  MoveL 1327 to (239.11, 156.17, 31.63) mm, rotated rx -180 ry 0 rz 180 deg; joints [-146.664, -89.82, -20.414, 62.265, 38.38, -56.149]
  MoveL 1328 to (239.11, 156.17, 31.63) mm, rotated rx -180 ry 0 rz 180 deg; joints [-146.664, -89.82, -20.414, 62.265, 38.38, -56.149]
  Call Extruder(256.49281)
  MoveL 1329 to (239, 156.42, 31.63) mm, rotated rx -180 ry 0 rz -180 deg; joints [-146.64, -89.832, -20.39, 62.3, 38.394, -56.183]
  MoveL 1330 to (239, 156.42, 31.63) mm, rotated rx -180 ry 0 rz -180 deg; joints [-146.64, -89.832, -20.39, 62.3, 38.394, -56.183]
  Call Extruder(256.65113)
  MoveL 1331 to (238.89, 156.66, 31.63) mm, rotated rx -180 ry 0 rz 180 deg; joints [-146.617, -89.843, -20.367, 62.335, 38.409, -56.217]
  MoveL 1332 to (238.89, 156.66, 31.63) mm, rotated rx -180 ry 0 rz 180 deg; joints [-146.617, -89.843, -20.367, 62.335, 38.409, -56.217]
  Call Extruder(256.83316)
  MoveL 1333 to (238.75, 156.94, 31.63) mm, rotated rx 180 ry 0 rz 180 deg; joints [-146.589, -89.851, -20.35, 62.369, 38.428, -56.249]
  MoveL 1334 to (238.75, 156.94, 31.63) mm, rotated rx 180 ry 0 rz 180 deg; joints [-146.589, -89.851, -20.35, 62.369, 38.428, -56.249]
  Call Extruder(257.03972)
  MoveL 1335 to (238.57, 157.25, 31.63) mm, rotated rx 180 ry 0 rz 180 deg; joints [-146.557, -89.857, -20.339, 62.403, 38.451, -56.278]
  MoveL 1336 to (238.57, 157.25, 31.63) mm, rotated rx 180 ry 0 rz 180 deg; joints [-146.557, -89.857, -20.339, 62.403, 38.451, -56.278]
  Call Extruder(257.24706)
  MoveL 1337 to (238.4, 157.55, 31.63) mm, rotated rx -180 ry 0 rz 180 deg; joints [-146.526, -89.862, -20.328, 62.437, 38.475, -56.308]
  MoveL 1338 to (238.4, 157.55, 31.63) mm, rotated rx -180 ry 0 rz 180 deg; joints [-146.526, -89.862, -20.328, 62.437, 38.475, -56.308]
  Call Extruder(257.45518)
  MoveL 1339 to (238.22, 157.85, 31.63) mm, rotated rx -180 ry 0 rz 180 deg; joints [-146.495, -89.867, -20.318, 62.471, 38.499, -56.338]
  MoveL 1340 to (238.22, 157.85, 31.63) mm, rotated rx -180 ry 0 rz 180 deg; joints [-146.495, -89.867, -20.318, 62.471, 38.499, -56.338]
  Call Extruder(257.57289)
  MoveL 1341 to (238.12, 158.03, 31.63) mm, rotated rx 180 ry 0 rz 180 deg; joints [-146.477, -89.87, -20.312, 62.49, 38.512, -56.354]
  MoveL 1342 to (238.12, 158.03, 31.63) mm, rotated rx 180 ry 0 rz 180 deg; joints [-146.477, -89.87, -20.312, 62.49, 38.512, -56.354]
  Call Extruder(257.90571)
  MoveL 1343 to (237.79, 158.48, 31.63) mm, rotated rx 180 ry 0 rz 180 deg; joints [-146.427, -89.864, -20.324, 62.528, 38.557, -56.38]
  MoveL 1344 to (237.79, 158.48, 31.63) mm, rotated rx 180 ry 0 rz 180 deg; joints [-146.427, -89.864, -20.324, 62.528, 38.557, -56.38]
  Call Extruder(258.23971)
  MoveL 1345 to (237.47, 158.93, 31.63) mm, rotated rx -180 ry 0 rz 180 deg; joints [-146.377, -89.858, -20.336, 62.566, 38.601, -56.406]
  MoveL 1346 to (237.47, 158.93, 31.63) mm, rotated rx -180 ry 0 rz 180 deg; joints [-146.377, -89.858, -20.336, 62.566, 38.601, -56.406]
  Call Extruder(258.40729)
  MoveL 1347 to (237.3, 159.15, 31.63) mm, rotated rx 180 ry 0 rz -180 deg; joints [-146.352, -89.855, -20.341, 62.585, 38.623, -56.419]
  Call Extruder(259.23663)
  MoveL 1348 to (236.39, 160.19, 31.63) mm, rotated rx 180 ry 0 rz 180 deg; joints [-146.229, -89.811, -20.432, 62.642, 38.747, -56.438]
  Call Extruder(259.86767)
  MoveL 1349 to (235.61, 160.89, 31.63) mm, rotated rx 180 ry 0 rz -180 deg; joints [-146.138, -89.747, -20.564, 62.648, 38.854, -56.406]
  MoveL 1350 to (235.61, 160.89, 31.63) mm, rotated rx 180 ry 0 rz -180 deg; joints [-146.138, -89.747, -20.564, 62.648, 38.854, -56.406]
  Call Extruder(260.06527)
  MoveL 1351 to (235.35, 161.1, 31.63) mm, rotated rx 180 ry 0 rz 180 deg; joints [-146.109, -89.725, -20.608, 62.648, 38.888, -56.394]
  Call Extruder(260.39930)
  MoveL 1352 to (234.9, 161.43, 31.63) mm, rotated rx 180 ry 0 rz -180 deg; joints [-146.062, -89.679, -20.702, 62.637, 38.949, -56.357]
  MoveL 1353 to (234.9, 161.43, 31.63) mm, rotated rx 180 ry 0 rz -180 deg; joints [-146.062, -89.679, -20.702, 62.637, 38.949, -56.357]
  Call Extruder(260.73214)
  MoveL 1354 to (234.45, 161.76, 31.63) mm, rotated rx 180 ry 0 rz 180 deg; joints [-146.015, -89.633, -20.796, 62.625, 39.01, -56.322]
  MoveL 1355 to (234.45, 161.76, 31.63) mm, rotated rx 180 ry 0 rz 180 deg; joints [-146.015, -89.633, -20.796, 62.625, 39.01, -56.322]
  Call Extruder(260.91134)
  MoveL 1356 to (234.21, 161.93, 31.63) mm, rotated rx -180 ry 0 rz 180 deg; joints [-145.99, -89.608, -20.848, 62.619, 39.044, -56.302]
  MoveL 1357 to (234.21, 161.93, 31.63) mm, rotated rx -180 ry 0 rz 180 deg; joints [-145.99, -89.608, -20.848, 62.619, 39.044, -56.302]
  Call Extruder(261.11946)
  MoveL 1358 to (233.9, 162.11, 31.63) mm, rotated rx 180 ry 0 rz 180 deg; joints [-145.961, -89.572, -20.923, 62.602, 39.085, -56.267]
  MoveL 1359 to (233.9, 162.11, 31.63) mm, rotated rx 180 ry 0 rz 180 deg; joints [-145.961, -89.572, -20.923, 62.602, 39.085, -56.267]
  Call Extruder(261.32679)
  MoveL 1360 to (233.6, 162.29, 31.63) mm, rotated rx 180 ry 0 rz 180 deg; joints [-145.933, -89.535, -20.998, 62.585, 39.126, -56.232]
  MoveL 1361 to (233.6, 162.29, 31.63) mm, rotated rx 180 ry 0 rz 180 deg; joints [-145.933, -89.535, -20.998, 62.585, 39.126, -56.232]
  Call Extruder(261.53335)
  MoveL 1362 to (233.29, 162.46, 31.63) mm, rotated rx -180 ry 0 rz -180 deg; joints [-145.905, -89.498, -21.073, 62.568, 39.167, -56.198]
  MoveL 1363 to (233.29, 162.46, 31.63) mm, rotated rx -180 ry 0 rz -180 deg; joints [-145.905, -89.498, -21.073, 62.568, 39.167, -56.198]
  Call Extruder(261.73913)
  MoveL 1364 to (232.99, 162.64, 31.63) mm, rotated rx 180 ry 0 rz -180 deg; joints [-145.876, -89.462, -21.147, 62.551, 39.209, -56.164]
  MoveL 1365 to (232.99, 162.64, 31.63) mm, rotated rx 180 ry 0 rz -180 deg; joints [-145.876, -89.462, -21.147, 62.551, 39.209, -56.164]
  Call Extruder(261.89741)
  MoveL 1366 to (232.74, 162.74, 31.63) mm, rotated rx -180 ry 0 rz 180 deg; joints [-145.856, -89.427, -21.218, 62.53, 39.242, -56.127]
  MoveL 1367 to (232.74, 162.74, 31.63) mm, rotated rx -180 ry 0 rz 180 deg; joints [-145.856, -89.427, -21.218, 62.53, 39.242, -56.127]
  Call Extruder(262.05508)
  MoveL 1368 to (232.49, 162.85, 31.63) mm, rotated rx 180 ry 0 rz -180 deg; joints [-145.835, -89.393, -21.289, 62.508, 39.276, -56.09]
  MoveL 1369 to (232.49, 162.85, 31.63) mm, rotated rx 180 ry 0 rz -180 deg; joints [-145.835, -89.393, -21.289, 62.508, 39.276, -56.09]
  Call Extruder(262.22517)
  MoveL 1370 to (232.22, 162.97, 31.63) mm, rotated rx 180 ry 0 rz 180 deg; joints [-145.813, -89.355, -21.366, 62.485, 39.313, -56.049]
  MoveL 1371 to (232.22, 162.97, 31.63) mm, rotated rx 180 ry 0 rz 180 deg; joints [-145.813, -89.355, -21.366, 62.485, 39.313, -56.049]
  Call Extruder(262.40753)
  MoveL 1372 to (231.93, 163.09, 31.63) mm, rotated rx -180 ry 0 rz 180 deg; joints [-145.789, -89.314, -21.45, 62.46, 39.352, -56.005]
  MoveL 1373 to (231.93, 163.09, 31.63) mm, rotated rx -180 ry 0 rz 180 deg; joints [-145.789, -89.314, -21.45, 62.46, 39.352, -56.005]
  Call Extruder(262.58914)
  MoveL 1374 to (231.64, 163.21, 31.63) mm, rotated rx -180 ry 0 rz 180 deg; joints [-145.766, -89.274, -21.534, 62.434, 39.392, -55.962]
  MoveL 1375 to (231.64, 163.21, 31.63) mm, rotated rx -180 ry 0 rz 180 deg; joints [-145.766, -89.274, -21.534, 62.434, 39.392, -55.962]
  Call Extruder(262.70258)
  MoveL 1376 to (231.45, 163.27, 31.63) mm, rotated rx 180 ry 0 rz -180 deg; joints [-145.751, -89.245, -21.592, 62.415, 39.417, -55.93]
  MoveL 1377 to (231.45, 163.27, 31.63) mm, rotated rx 180 ry 0 rz -180 deg; joints [-145.751, -89.245, -21.592, 62.415, 39.417, -55.93]
  Call Extruder(262.81558)
  MoveL 1378 to (231.26, 163.33, 31.63) mm, rotated rx 180 ry 0 rz 180 deg; joints [-145.737, -89.217, -21.65, 62.395, 39.443, -55.898]
  MoveL 1379 to (231.26, 163.33, 31.63) mm, rotated rx 180 ry 0 rz 180 deg; joints [-145.737, -89.217, -21.65, 62.395, 39.443, -55.898]
  Call Extruder(262.92814)
  MoveL 1380 to (231.07, 163.39, 31.63) mm, rotated rx -180 ry 0 rz -180 deg; joints [-145.723, -89.189, -21.708, 62.375, 39.468, -55.866]
  MoveL 1381 to (231.07, 163.39, 31.63) mm, rotated rx -180 ry 0 rz -180 deg; joints [-145.723, -89.189, -21.708, 62.375, 39.468, -55.866]
  Call Extruder(263.04025)
  MoveL 1382 to (230.88, 163.45, 31.63) mm, rotated rx 180 ry 0 rz 180 deg; joints [-145.709, -89.16, -21.766, 62.356, 39.494, -55.834]
  MoveL 1383 to (230.88, 163.45, 31.63) mm, rotated rx 180 ry 0 rz 180 deg; joints [-145.709, -89.16, -21.766, 62.356, 39.494, -55.834]
  Call Extruder(263.15191)
  MoveL 1384 to (230.7, 163.51, 31.63) mm, rotated rx 180 ry 0 rz -180 deg; joints [-145.695, -89.132, -21.824, 62.336, 39.519, -55.802]
  MoveL 1385 to (230.7, 163.51, 31.63) mm, rotated rx 180 ry 0 rz -180 deg; joints [-145.695, -89.132, -21.824, 62.336, 39.519, -55.802]
  Call Extruder(263.28301)
  MoveL 1386 to (230.47, 163.58, 31.63) mm, rotated rx 180 ry 0 rz 180 deg; joints [-145.679, -89.098, -21.894, 62.312, 39.55, -55.764]
  MoveL 1387 to (230.47, 163.58, 31.63) mm, rotated rx 180 ry 0 rz 180 deg; joints [-145.679, -89.098, -21.894, 62.312, 39.55, -55.764]
  Call Extruder(263.41354)
  MoveL 1388 to (230.25, 163.65, 31.63) mm, rotated rx -180 ry 0 rz 180 deg; joints [-145.662, -89.064, -21.964, 62.288, 39.58, -55.725]
  MoveL 1389 to (230.25, 163.65, 31.63) mm, rotated rx -180 ry 0 rz 180 deg; joints [-145.662, -89.064, -21.964, 62.288, 39.58, -55.725]
  Call Extruder(263.54350)
  MoveL 1390 to (230.02, 163.72, 31.63) mm, rotated rx 180 ry 0 rz 180 deg; joints [-145.646, -89.031, -22.033, 62.265, 39.61, -55.687]
  MoveL 1391 to (230.02, 163.72, 31.63) mm, rotated rx 180 ry 0 rz 180 deg; joints [-145.646, -89.031, -22.033, 62.265, 39.61, -55.687]
  Call Extruder(263.67290)
  MoveL 1392 to (229.8, 163.78, 31.63) mm, rotated rx -180 ry 0 rz 180 deg; joints [-145.629, -88.997, -22.102, 62.241, 39.64, -55.648]
  MoveL 1393 to (229.8, 163.78, 31.63) mm, rotated rx -180 ry 0 rz 180 deg; joints [-145.629, -88.997, -22.102, 62.241, 39.64, -55.648]
  Call Extruder(263.79488)
  MoveL 1394 to (229.59, 163.84, 31.63) mm, rotated rx 180 ry 0 rz -180 deg; joints [-145.614, -88.964, -22.171, 62.217, 39.669, -55.61]
  MoveL 1395 to (229.59, 163.84, 31.63) mm, rotated rx 180 ry 0 rz -180 deg; joints [-145.614, -88.964, -22.171, 62.217, 39.669, -55.61]
  Call Extruder(263.90973)
  MoveL 1396 to (229.38, 163.88, 31.63) mm, rotated rx 180 ry 0 rz -180 deg; joints [-145.601, -88.931, -22.238, 62.192, 39.696, -55.571]
  MoveL 1397 to (229.38, 163.88, 31.63) mm, rotated rx 180 ry 0 rz -180 deg; joints [-145.601, -88.931, -22.238, 62.192, 39.696, -55.571]
  Call Extruder(264.02412)
  MoveL 1398 to (229.18, 163.93, 31.63) mm, rotated rx 180 ry 0 rz -180 deg; joints [-145.587, -88.898, -22.306, 62.167, 39.724, -55.533]
  MoveL 1399 to (229.18, 163.93, 31.63) mm, rotated rx 180 ry 0 rz -180 deg; joints [-145.587, -88.898, -22.306, 62.167, 39.724, -55.533]
  Call Extruder(264.13806)
  MoveL 1400 to (228.97, 163.97, 31.63) mm, rotated rx 180 ry 0 rz 180 deg; joints [-145.573, -88.865, -22.373, 62.143, 39.751, -55.494]
  MoveL 1401 to (228.97, 163.97, 31.63) mm, rotated rx 180 ry 0 rz 180 deg; joints [-145.573, -88.865, -22.373, 62.143, 39.751, -55.494]
  Call Extruder(264.25155)
  MoveL 1402 to (228.77, 164.02, 31.63) mm, rotated rx -180 ry 0 rz 180 deg; joints [-145.559, -88.833, -22.44, 62.118, 39.779, -55.456]
  MoveL 1403 to (228.77, 164.02, 31.63) mm, rotated rx -180 ry 0 rz 180 deg; joints [-145.559, -88.833, -22.44, 62.118, 39.779, -55.456]
  Call Extruder(264.38884)
  MoveL 1404 to (228.52, 164.07, 31.63) mm, rotated rx -180 ry 0 rz -180 deg; joints [-145.543, -88.792, -22.523, 62.088, 39.812, -55.408]
  MoveL 1405 to (228.52, 164.07, 31.63) mm, rotated rx -180 ry 0 rz -180 deg; joints [-145.543, -88.792, -22.523, 62.088, 39.812, -55.408]
  Call Extruder(264.52551)
  MoveL 1406 to (228.27, 164.12, 31.63) mm, rotated rx -180 ry 0 rz 180 deg; joints [-145.527, -88.752, -22.606, 62.057, 39.846, -55.36]
  MoveL 1407 to (228.27, 164.12, 31.63) mm, rotated rx -180 ry 0 rz 180 deg; joints [-145.527, -88.752, -22.606, 62.057, 39.846, -55.36]
  Call Extruder(264.66157)
  MoveL 1408 to (228.02, 164.17, 31.63) mm, rotated rx -180 ry 0 rz -180 deg; joints [-145.51, -88.712, -22.689, 62.027, 39.879, -55.313]
  MoveL 1409 to (228.02, 164.17, 31.63) mm, rotated rx -180 ry 0 rz -180 deg; joints [-145.51, -88.712, -22.689, 62.027, 39.879, -55.313]
  Call Extruder(264.79703)
  MoveL 1410 to (227.77, 164.22, 31.63) mm, rotated rx 180 ry 0 rz -180 deg; joints [-145.494, -88.672, -22.771, 61.996, 39.913, -55.266]
  MoveL 1411 to (227.77, 164.22, 31.63) mm, rotated rx 180 ry 0 rz -180 deg; joints [-145.494, -88.672, -22.771, 61.996, 39.913, -55.266]
  Call Extruder(264.93187)
  MoveL 1412 to (227.52, 164.27, 31.63) mm, rotated rx 180 ry 0 rz -180 deg; joints [-145.477, -88.632, -22.853, 61.966, 39.946, -55.219]
  MoveL 1413 to (227.52, 164.27, 31.63) mm, rotated rx 180 ry 0 rz -180 deg; joints [-145.477, -88.632, -22.853, 61.966, 39.946, -55.219]
  Call Extruder(265.06610)
  MoveL 1414 to (227.27, 164.32, 31.63) mm, rotated rx -180 ry 0 rz 180 deg; joints [-145.461, -88.593, -22.935, 61.937, 39.979, -55.172]
  MoveL 1415 to (227.27, 164.32, 31.63) mm, rotated rx -180 ry 0 rz 180 deg; joints [-145.461, -88.593, -22.935, 61.937, 39.979, -55.172]
  Call Extruder(265.19972)
  MoveL 1416 to (227.02, 164.37, 31.63) mm, rotated rx 180 ry 0 rz -180 deg; joints [-145.444, -88.553, -23.017, 61.907, 40.013, -55.125]
  MoveL 1417 to (227.02, 164.37, 31.63) mm, rotated rx 180 ry 0 rz -180 deg; joints [-145.444, -88.553, -23.017, 61.907, 40.013, -55.125]
  Call Extruder(265.36183)
  MoveL 1418 to (226.72, 164.41, 31.63) mm, rotated rx -180 ry 0 rz 180 deg; joints [-145.425, -88.503, -23.12, 61.868, 40.054, -55.066]
  MoveL 1419 to (226.72, 164.41, 31.63) mm, rotated rx -180 ry 0 rz 180 deg; joints [-145.425, -88.503, -23.12, 61.868, 40.054, -55.066]
  Call Extruder(265.52320)
  MoveL 1420 to (226.41, 164.46, 31.63) mm, rotated rx 180 ry 0 rz 180 deg; joints [-145.406, -88.453, -23.223, 61.83, 40.094, -55.006]
  MoveL 1421 to (226.41, 164.46, 31.63) mm, rotated rx 180 ry 0 rz 180 deg; joints [-145.406, -88.453, -23.223, 61.83, 40.094, -55.006]
  Call Extruder(265.68385)
  MoveL 1422 to (226.11, 164.51, 31.63) mm, rotated rx 180 ry 0 rz 180 deg; joints [-145.386, -88.403, -23.326, 61.792, 40.135, -54.947]
  MoveL 1423 to (226.11, 164.51, 31.63) mm, rotated rx 180 ry 0 rz 180 deg; joints [-145.386, -88.403, -23.326, 61.792, 40.135, -54.947]
  Call Extruder(265.84377)
  MoveL 1424 to (225.8, 164.56, 31.63) mm, rotated rx -180 ry 0 rz 180 deg; joints [-145.367, -88.354, -23.428, 61.754, 40.176, -54.888]
  MoveL 1425 to (225.8, 164.56, 31.63) mm, rotated rx -180 ry 0 rz 180 deg; joints [-145.367, -88.354, -23.428, 61.754, 40.176, -54.888]
  Call Extruder(266.00296)
  MoveL 1426 to (225.5, 164.61, 31.63) mm, rotated rx 180 ry 0 rz 180 deg; joints [-145.348, -88.304, -23.53, 61.717, 40.217, -54.83]
  MoveL 1427 to (225.5, 164.61, 31.63) mm, rotated rx 180 ry 0 rz 180 deg; joints [-145.348, -88.304, -23.53, 61.717, 40.217, -54.83]
  Call Extruder(266.16143)
  MoveL 1428 to (225.19, 164.66, 31.63) mm, rotated rx -180 ry 0 rz -180 deg; joints [-145.328, -88.255, -23.632, 61.679, 40.258, -54.771]
  MoveL 1429 to (225.19, 164.66, 31.63) mm, rotated rx -180 ry 0 rz -180 deg; joints [-145.328, -88.255, -23.632, 61.679, 40.258, -54.771]
  Call Extruder(266.36030)
  MoveL 1430 to (224.8, 164.7, 31.63) mm, rotated rx -180 ry 0 rz 180 deg; joints [-145.305, -88.191, -23.764, 61.629, 40.309, -54.694]
  MoveL 1431 to (224.8, 164.7, 31.63) mm, rotated rx -180 ry 0 rz 180 deg; joints [-145.305, -88.191, -23.764, 61.629, 40.309, -54.694]
  Call Extruder(266.55831)
  MoveL 1432 to (224.42, 164.75, 31.63) mm, rotated rx -180 ry 0 rz 180 deg; joints [-145.281, -88.127, -23.896, 61.58, 40.361, -54.618]
  MoveL 1433 to (224.42, 164.75, 31.63) mm, rotated rx -180 ry 0 rz 180 deg; joints [-145.281, -88.127, -23.896, 61.58, 40.361, -54.618]
  Call Extruder(266.75545)
  MoveL 1434 to (224.03, 164.79, 31.63) mm, rotated rx 180 ry 0 rz 180 deg; joints [-145.258, -88.064, -24.027, 61.53, 40.412, -54.542]
  MoveL 1435 to (224.03, 164.79, 31.63) mm, rotated rx 180 ry 0 rz 180 deg; joints [-145.258, -88.064, -24.027, 61.53, 40.412, -54.542]
  Call Extruder(266.95173)
  MoveL 1436 to (223.64, 164.84, 31.63) mm, rotated rx -180 ry 0 rz 180 deg; joints [-145.234, -88, -24.158, 61.482, 40.463, -54.466]
  MoveL 1437 to (223.64, 164.84, 31.63) mm, rotated rx -180 ry 0 rz 180 deg; joints [-145.234, -88, -24.158, 61.482, 40.463, -54.466]
  Call Extruder(267.19740)
  MoveL 1438 to (223.15, 164.89, 31.63) mm, rotated rx 180 ry 0 rz 180 deg; joints [-145.206, -87.92, -24.325, 61.419, 40.528, -54.369]
  MoveL 1439 to (223.15, 164.89, 31.63) mm, rotated rx 180 ry 0 rz 180 deg; joints [-145.206, -87.92, -24.325, 61.419, 40.528, -54.369]
  Call Extruder(267.49209)
  MoveL 1440 to (222.56, 164.93, 31.63) mm, rotated rx -180 ry 0 rz 180 deg; joints [-145.172, -87.821, -24.528, 61.341, 40.606, -54.25]
  MoveL 1441 to (222.56, 164.93, 31.63) mm, rotated rx -180 ry 0 rz 180 deg; joints [-145.172, -87.821, -24.528, 61.341, 40.606, -54.25]
  Call Extruder(267.78545)
  MoveL 1442 to (221.97, 164.98, 31.63) mm, rotated rx 180 ry 0 rz -180 deg; joints [-145.138, -87.724, -24.73, 61.265, 40.684, -54.133]
  MoveL 1443 to (221.97, 164.98, 31.63) mm, rotated rx 180 ry 0 rz -180 deg; joints [-145.138, -87.724, -24.73, 61.265, 40.684, -54.133]
  Call Extruder(268.21876)
  MoveL 1444 to (221.1, 165.02, 31.63) mm, rotated rx -180 ry 0 rz 180 deg; joints [-145.088, -87.578, -25.034, 61.15, 40.799, -53.955]
  MoveL 1445 to (221.1, 165.02, 31.63) mm, rotated rx -180 ry 0 rz 180 deg; joints [-145.088, -87.578, -25.034, 61.15, 40.799, -53.955]
  Call Extruder(268.79092)
  MoveL 1446 to (219.94, 165.07, 31.63) mm, rotated rx 180 ry 0 rz -180 deg; joints [-145.024, -87.384, -25.436, 60.996, 40.952, -53.72]
  MoveL 1447 to (219.94, 165.07, 31.63) mm, rotated rx 180 ry 0 rz -180 deg; joints [-145.024, -87.384, -25.436, 60.996, 40.952, -53.72]
  Call Extruder(269.21879)
  MoveL 1448 to (219.06, 165.09, 31.63) mm, rotated rx -180 ry 0 rz -180 deg; joints [-144.977, -87.238, -25.74, 60.88, 41.066, -53.542]
  Call Extruder(385.86744)
  MoveL 1449 to (-19.06, 165.09, 31.63) mm, rotated rx -180 ry 0 rz -180 deg; joints [-127.435, -66.78, -72.976, 59.702, 66.877, -33.904]
  MoveL 1450 to (-19.06, 165.09, 31.63) mm, rotated rx -180 ry 0 rz -180 deg; joints [-127.435, -66.78, -72.976, 59.702, 66.877, -33.904]
  Call Extruder(386.58306)
  MoveL 1451 to (-20.52, 165.05, 31.63) mm, rotated rx -180 ry 0 rz 180 deg; joints [-127.291, -66.713, -73.159, 59.788, 67.016, -33.846]
  MoveL 1452 to (-20.52, 165.05, 31.63) mm, rotated rx -180 ry 0 rz 180 deg; joints [-127.291, -66.713, -73.159, 59.788, 67.016, -33.846]
  Call Extruder(387.15780)
  MoveL 1453 to (-21.68, 165, 31.63) mm, rotated rx -180 ry 0 rz 180 deg; joints [-127.178, -66.659, -73.307, 59.856, 67.126, -33.797]
  MoveL 1454 to (-21.68, 165, 31.63) mm, rotated rx -180 ry 0 rz 180 deg; joints [-127.178, -66.659, -73.307, 59.856, 67.126, -33.797]
  Call Extruder(387.45117)
  MoveL 1455 to (-22.27, 164.95, 31.63) mm, rotated rx -180 ry 0 rz -180 deg; joints [-127.122, -66.63, -73.386, 59.889, 67.182, -33.77]
  MoveL 1456 to (-22.27, 164.95, 31.63) mm, rotated rx -180 ry 0 rz -180 deg; joints [-127.122, -66.63, -73.386, 59.889, 67.182, -33.77]
  Call Extruder(387.74586)
  MoveL 1457 to (-22.86, 164.91, 31.63) mm, rotated rx 180 ry 0 rz -180 deg; joints [-127.065, -66.602, -73.464, 59.921, 67.239, -33.743]
  MoveL 1458 to (-22.86, 164.91, 31.63) mm, rotated rx 180 ry 0 rz -180 deg; joints [-127.065, -66.602, -73.464, 59.921, 67.239, -33.743]
  Call Extruder(388.04189)
  MoveL 1459 to (-23.45, 164.86, 31.63) mm, rotated rx 180 ry 0 rz 180 deg; joints [-127.009, -66.573, -73.542, 59.954, 67.295, -33.716]
  MoveL 1460 to (-23.45, 164.86, 31.63) mm, rotated rx 180 ry 0 rz 180 deg; joints [-127.009, -66.573, -73.542, 59.954, 67.295, -33.716]
  Call Extruder(388.23816)
  MoveL 1461 to (-23.84, 164.82, 31.63) mm, rotated rx 180 ry 0 rz 180 deg; joints [-126.973, -66.554, -73.596, 59.974, 67.332, -33.696]
  MoveL 1462 to (-23.84, 164.82, 31.63) mm, rotated rx 180 ry 0 rz 180 deg; joints [-126.973, -66.554, -73.596, 59.974, 67.332, -33.696]
  Call Extruder(388.43530)
  MoveL 1463 to (-24.22, 164.77, 31.63) mm, rotated rx 180 ry 0 rz 180 deg; joints [-126.937, -66.535, -73.649, 59.994, 67.369, -33.676]
  MoveL 1464 to (-24.22, 164.77, 31.63) mm, rotated rx 180 ry 0 rz 180 deg; joints [-126.937, -66.535, -73.649, 59.994, 67.369, -33.676]
  Call Extruder(388.63331)
  MoveL 1465 to (-24.61, 164.72, 31.63) mm, rotated rx -180 ry 0 rz 180 deg; joints [-126.901, -66.515, -73.703, 60.014, 67.406, -33.657]
  MoveL 1466 to (-24.61, 164.72, 31.63) mm, rotated rx -180 ry 0 rz 180 deg; joints [-126.901, -66.515, -73.703, 60.014, 67.406, -33.657]
  Call Extruder(388.83219)
  MoveL 1467 to (-25, 164.68, 31.63) mm, rotated rx 180 ry 0 rz 180 deg; joints [-126.865, -66.496, -73.757, 60.034, 67.443, -33.637]
  MoveL 1468 to (-25, 164.68, 31.63) mm, rotated rx 180 ry 0 rz 180 deg; joints [-126.865, -66.496, -73.757, 60.034, 67.443, -33.637]
  Call Extruder(389.01127)
  MoveL 1469 to (-25.34, 164.63, 31.63) mm, rotated rx -180 ry 0 rz -180 deg; joints [-126.834, -66.478, -73.805, 60.051, 67.476, -33.619]
  MoveL 1470 to (-25.34, 164.63, 31.63) mm, rotated rx -180 ry 0 rz -180 deg; joints [-126.834, -66.478, -73.805, 60.051, 67.476, -33.619]
  Call Extruder(389.17046)
  MoveL 1471 to (-25.65, 164.58, 31.63) mm, rotated rx -180 ry 0 rz -180 deg; joints [-126.806, -66.462, -73.85, 60.066, 67.505, -33.602]
  MoveL 1472 to (-25.65, 164.58, 31.63) mm, rotated rx -180 ry 0 rz -180 deg; joints [-126.806, -66.462, -73.85, 60.066, 67.505, -33.602]
  Call Extruder(389.33039)
  MoveL 1473 to (-25.96, 164.53, 31.63) mm, rotated rx 180 ry 0 rz 180 deg; joints [-126.779, -66.446, -73.894, 60.081, 67.535, -33.585]
  MoveL 1474 to (-25.96, 164.53, 31.63) mm, rotated rx 180 ry 0 rz 180 deg; joints [-126.779, -66.446, -73.894, 60.081, 67.535, -33.585]
  Call Extruder(389.49104)
  MoveL 1475 to (-26.26, 164.49, 31.63) mm, rotated rx -180 ry 0 rz 180 deg; joints [-126.751, -66.43, -73.938, 60.096, 67.564, -33.568]
  MoveL 1476 to (-26.26, 164.49, 31.63) mm, rotated rx -180 ry 0 rz 180 deg; joints [-126.751, -66.43, -73.938, 60.096, 67.564, -33.568]
  Call Extruder(389.65242)
  MoveL 1477 to (-26.57, 164.44, 31.63) mm, rotated rx 180 ry 0 rz 180 deg; joints [-126.723, -66.414, -73.982, 60.111, 67.593, -33.551]
  MoveL 1478 to (-26.57, 164.44, 31.63) mm, rotated rx 180 ry 0 rz 180 deg; joints [-126.723, -66.414, -73.982, 60.111, 67.593, -33.551]
  Call Extruder(389.81452)
  MoveL 1479 to (-26.87, 164.39, 31.63) mm, rotated rx -180 ry 0 rz 180 deg; joints [-126.696, -66.399, -74.026, 60.125, 67.622, -33.534]
  MoveL 1480 to (-26.87, 164.39, 31.63) mm, rotated rx -180 ry 0 rz 180 deg; joints [-126.696, -66.399, -74.026, 60.125, 67.622, -33.534]
  Call Extruder(389.96273)
  MoveL 1481 to (-27.15, 164.34, 31.63) mm, rotated rx 180 ry 0 rz 180 deg; joints [-126.671, -66.384, -74.066, 60.138, 67.649, -33.519]
  MoveL 1482 to (-27.15, 164.34, 31.63) mm, rotated rx 180 ry 0 rz 180 deg; joints [-126.671, -66.384, -74.066, 60.138, 67.649, -33.519]
  Call Extruder(390.09696)
  MoveL 1483 to (-27.4, 164.29, 31.63) mm, rotated rx 180 ry 0 rz 180 deg; joints [-126.649, -66.37, -74.104, 60.149, 67.673, -33.504]
  MoveL 1484 to (-27.4, 164.29, 31.63) mm, rotated rx 180 ry 0 rz 180 deg; joints [-126.649, -66.37, -74.104, 60.149, 67.673, -33.504]
  Call Extruder(390.23180)
  MoveL 1485 to (-27.65, 164.24, 31.63) mm, rotated rx -180 ry 0 rz -180 deg; joints [-126.628, -66.357, -74.141, 60.161, 67.697, -33.489]
  MoveL 1486 to (-27.65, 164.24, 31.63) mm, rotated rx -180 ry 0 rz -180 deg; joints [-126.628, -66.357, -74.141, 60.161, 67.697, -33.489]
  Call Extruder(390.36725)
  MoveL 1487 to (-27.9, 164.19, 31.63) mm, rotated rx 180 ry 0 rz 180 deg; joints [-126.606, -66.344, -74.178, 60.172, 67.721, -33.474]
  MoveL 1488 to (-27.9, 164.19, 31.63) mm, rotated rx 180 ry 0 rz 180 deg; joints [-126.606, -66.344, -74.178, 60.172, 67.721, -33.474]
  Call Extruder(390.50331)
  MoveL 1489 to (-28.15, 164.14, 31.63) mm, rotated rx 180 ry 0 rz -180 deg; joints [-126.584, -66.33, -74.216, 60.183, 67.745, -33.459]
  MoveL 1490 to (-28.15, 164.14, 31.63) mm, rotated rx 180 ry 0 rz -180 deg; joints [-126.584, -66.33, -74.216, 60.183, 67.745, -33.459]
  Call Extruder(390.63999)
  MoveL 1491 to (-28.4, 164.09, 31.63) mm, rotated rx 180 ry 0 rz 180 deg; joints [-126.562, -66.317, -74.253, 60.194, 67.769, -33.444]
  MoveL 1492 to (-28.4, 164.09, 31.63) mm, rotated rx 180 ry 0 rz 180 deg; joints [-126.562, -66.317, -74.253, 60.194, 67.769, -33.444]
  Call Extruder(390.77727)
  MoveL 1493 to (-28.64, 164.04, 31.63) mm, rotated rx 180 ry 0 rz 180 deg; joints [-126.54, -66.303, -74.29, 60.206, 67.792, -33.429]
  MoveL 1494 to (-28.64, 164.04, 31.63) mm, rotated rx 180 ry 0 rz 180 deg; joints [-126.54, -66.303, -74.29, 60.206, 67.792, -33.429]
  Call Extruder(390.90294)
  MoveL 1495 to (-28.87, 164, 31.63) mm, rotated rx 180 ry 0 rz 180 deg; joints [-126.52, -66.291, -74.324, 60.216, 67.814, -33.415]
  MoveL 1496 to (-28.87, 164, 31.63) mm, rotated rx 180 ry 0 rz 180 deg; joints [-126.52, -66.291, -74.324, 60.216, 67.814, -33.415]
  Call Extruder(391.01688)
  MoveL 1497 to (-29.08, 163.95, 31.63) mm, rotated rx 180 ry 0 rz 180 deg; joints [-126.503, -66.28, -74.355, 60.224, 67.834, -33.403]
  MoveL 1498 to (-29.08, 163.95, 31.63) mm, rotated rx 180 ry 0 rz 180 deg; joints [-126.503, -66.28, -74.355, 60.224, 67.834, -33.403]
  Call Extruder(391.13127)
  MoveL 1499 to (-29.28, 163.91, 31.63) mm, rotated rx 180 ry 0 rz 180 deg; joints [-126.485, -66.269, -74.386, 60.233, 67.853, -33.39]
  MoveL 1500 to (-29.28, 163.91, 31.63) mm, rotated rx 180 ry 0 rz 180 deg; joints [-126.485, -66.269, -74.386, 60.233, 67.853, -33.39]
  Call Extruder(391.24612)
  MoveL 1501 to (-29.48, 163.86, 31.63) mm, rotated rx 180 ry 0 rz 180 deg; joints [-126.467, -66.258, -74.417, 60.242, 67.873, -33.377]
  MoveL 1502 to (-29.48, 163.86, 31.63) mm, rotated rx 180 ry 0 rz 180 deg; joints [-126.467, -66.258, -74.417, 60.242, 67.873, -33.377]
  Call Extruder(391.36141)
  MoveL 1503 to (-29.69, 163.82, 31.63) mm, rotated rx 180 ry 0 rz 180 deg; joints [-126.45, -66.246, -74.449, 60.251, 67.893, -33.365]
  MoveL 1504 to (-29.69, 163.82, 31.63) mm, rotated rx 180 ry 0 rz 180 deg; joints [-126.45, -66.246, -74.449, 60.251, 67.893, -33.365]
  Call Extruder(391.49081)
  MoveL 1505 to (-29.91, 163.75, 31.63) mm, rotated rx -180 ry 0 rz 180 deg; joints [-126.432, -66.233, -74.485, 60.259, 67.914, -33.349]
  MoveL 1506 to (-29.91, 163.75, 31.63) mm, rotated rx -180 ry 0 rz 180 deg; joints [-126.432, -66.233, -74.485, 60.259, 67.914, -33.349]
  Call Extruder(391.62077)
  MoveL 1507 to (-30.14, 163.68, 31.63) mm, rotated rx 180 ry 0 rz 180 deg; joints [-126.414, -66.22, -74.522, 60.267, 67.936, -33.332]
  MoveL 1508 to (-30.14, 163.68, 31.63) mm, rotated rx 180 ry 0 rz 180 deg; joints [-126.414, -66.22, -74.522, 60.267, 67.936, -33.332]
  Call Extruder(391.75130)
  MoveL 1509 to (-30.36, 163.61, 31.63) mm, rotated rx 180 ry 0 rz 180 deg; joints [-126.396, -66.207, -74.559, 60.275, 67.958, -33.316]
  MoveL 1510 to (-30.36, 163.61, 31.63) mm, rotated rx 180 ry 0 rz 180 deg; joints [-126.396, -66.207, -74.559, 60.275, 67.958, -33.316]
  Call Extruder(391.88239)
  MoveL 1511 to (-30.58, 163.55, 31.63) mm, rotated rx 180 ry 0 rz 180 deg; joints [-126.378, -66.194, -74.596, 60.283, 67.979, -33.3]
  MoveL 1512 to (-30.58, 163.55, 31.63) mm, rotated rx 180 ry 0 rz 180 deg; joints [-126.378, -66.194, -74.596, 60.283, 67.979, -33.3]
  Call Extruder(392.00403)
  MoveL 1513 to (-30.79, 163.48, 31.63) mm, rotated rx 180 ry 0 rz 180 deg; joints [-126.361, -66.181, -74.631, 60.29, 67.999, -33.285]
  MoveL 1514 to (-30.79, 163.48, 31.63) mm, rotated rx 180 ry 0 rz 180 deg; joints [-126.361, -66.181, -74.631, 60.29, 67.999, -33.285]
  Call Extruder(392.11615)
  MoveL 1515 to (-30.98, 163.42, 31.63) mm, rotated rx 180 ry 0 rz -180 deg; joints [-126.347, -66.17, -74.662, 60.296, 68.017, -33.271]
  MoveL 1516 to (-30.98, 163.42, 31.63) mm, rotated rx 180 ry 0 rz -180 deg; joints [-126.347, -66.17, -74.662, 60.296, 68.017, -33.271]
  Call Extruder(392.22871)
  MoveL 1517 to (-31.17, 163.36, 31.63) mm, rotated rx 180 ry 0 rz -180 deg; joints [-126.332, -66.159, -74.694, 60.302, 68.036, -33.257]
  MoveL 1518 to (-31.17, 163.36, 31.63) mm, rotated rx 180 ry 0 rz -180 deg; joints [-126.332, -66.159, -74.694, 60.302, 68.036, -33.257]
  Call Extruder(392.34171)
  MoveL 1519 to (-31.35, 163.3, 31.63) mm, rotated rx 180 ry 0 rz 180 deg; joints [-126.317, -66.147, -74.726, 60.309, 68.054, -33.243]
  MoveL 1520 to (-31.35, 163.3, 31.63) mm, rotated rx 180 ry 0 rz 180 deg; joints [-126.317, -66.147, -74.726, 60.309, 68.054, -33.243]
  Call Extruder(392.45516)
  MoveL 1521 to (-31.54, 163.24, 31.63) mm, rotated rx 180 ry 0 rz 180 deg; joints [-126.302, -66.136, -74.757, 60.315, 68.072, -33.229]
  MoveL 1522 to (-31.54, 163.24, 31.63) mm, rotated rx 180 ry 0 rz 180 deg; joints [-126.302, -66.136, -74.757, 60.315, 68.072, -33.229]
  Call Extruder(392.60280)
  MoveL 1523 to (-31.78, 163.15, 31.63) mm, rotated rx 180 ry 0 rz 180 deg; joints [-126.284, -66.121, -74.8, 60.322, 68.095, -33.209]
  MoveL 1524 to (-31.78, 163.15, 31.63) mm, rotated rx 180 ry 0 rz 180 deg; joints [-126.284, -66.121, -74.8, 60.322, 68.095, -33.209]
  Call Extruder(392.78516)
  MoveL 1525 to (-32.07, 163.03, 31.63) mm, rotated rx 180 ry 0 rz 180 deg; joints [-126.263, -66.102, -74.853, 60.329, 68.124, -33.185]
  MoveL 1526 to (-32.07, 163.03, 31.63) mm, rotated rx 180 ry 0 rz 180 deg; joints [-126.263, -66.102, -74.853, 60.329, 68.124, -33.185]
  Call Extruder(392.96827)
  MoveL 1527 to (-32.37, 162.91, 31.63) mm, rotated rx 180 ry 0 rz 180 deg; joints [-126.241, -66.083, -74.906, 60.336, 68.152, -33.16]
  MoveL 1528 to (-32.37, 162.91, 31.63) mm, rotated rx 180 ry 0 rz 180 deg; joints [-126.241, -66.083, -74.906, 60.336, 68.152, -33.16]
  Call Extruder(393.12594)
  MoveL 1529 to (-32.62, 162.8, 31.63) mm, rotated rx 180 ry 0 rz 180 deg; joints [-126.224, -66.067, -74.952, 60.342, 68.177, -33.138]
  MoveL 1530 to (-32.62, 162.8, 31.63) mm, rotated rx 180 ry 0 rz 180 deg; joints [-126.224, -66.067, -74.952, 60.342, 68.177, -33.138]
  Call Extruder(393.28422)
  MoveL 1531 to (-32.86, 162.69, 31.63) mm, rotated rx 180 ry 0 rz 180 deg; joints [-126.206, -66.05, -74.998, 60.348, 68.201, -33.117]
  MoveL 1532 to (-32.86, 162.69, 31.63) mm, rotated rx 180 ry 0 rz 180 deg; joints [-126.206, -66.05, -74.998, 60.348, 68.201, -33.117]
  Call Extruder(393.46623)
  MoveL 1533 to (-33.14, 162.55, 31.63) mm, rotated rx 180 ry 0 rz 180 deg; joints [-126.188, -66.031, -75.052, 60.352, 68.228, -33.09]
  MoveL 1534 to (-33.14, 162.55, 31.63) mm, rotated rx 180 ry 0 rz 180 deg; joints [-126.188, -66.031, -75.052, 60.352, 68.228, -33.09]
  Call Extruder(393.67279)
  MoveL 1535 to (-33.45, 162.37, 31.63) mm, rotated rx 180 ry 0 rz -180 deg; joints [-126.169, -66.008, -75.115, 60.354, 68.258, -33.058]
  MoveL 1536 to (-33.45, 162.37, 31.63) mm, rotated rx 180 ry 0 rz -180 deg; joints [-126.169, -66.008, -75.115, 60.354, 68.258, -33.058]
  Call Extruder(393.88012)
  MoveL 1537 to (-33.75, 162.2, 31.63) mm, rotated rx 180 ry 0 rz 180 deg; joints [-126.151, -65.986, -75.178, 60.357, 68.288, -33.026]
  MoveL 1538 to (-33.75, 162.2, 31.63) mm, rotated rx 180 ry 0 rz 180 deg; joints [-126.151, -65.986, -75.178, 60.357, 68.288, -33.026]
  Call Extruder(394.08824)
  MoveL 1539 to (-34.05, 162.02, 31.63) mm, rotated rx 180 ry 0 rz 180 deg; joints [-126.133, -65.964, -75.241, 60.359, 68.319, -32.994]
  MoveL 1540 to (-34.05, 162.02, 31.63) mm, rotated rx 180 ry 0 rz 180 deg; joints [-126.133, -65.964, -75.241, 60.359, 68.319, -32.994]
  Call Extruder(394.20594)
  MoveL 1541 to (-34.23, 161.92, 31.63) mm, rotated rx -180 ry 0 rz -180 deg; joints [-126.122, -65.951, -75.276, 60.361, 68.335, -32.976]
  MoveL 1542 to (-34.23, 161.92, 31.63) mm, rotated rx -180 ry 0 rz -180 deg; joints [-126.122, -65.951, -75.276, 60.361, 68.335, -32.976]
  Call Extruder(394.53878)
  MoveL 1543 to (-34.68, 161.59, 31.63) mm, rotated rx 180 ry 0 rz 180 deg; joints [-126.1, -65.914, -75.38, 60.358, 68.381, -32.921]
  MoveL 1544 to (-34.68, 161.59, 31.63) mm, rotated rx 180 ry 0 rz 180 deg; joints [-126.1, -65.914, -75.38, 60.358, 68.381, -32.921]
  Call Extruder(394.87281)
  MoveL 1545 to (-35.13, 161.27, 31.63) mm, rotated rx 180 ry 0 rz 180 deg; joints [-126.078, -65.877, -75.484, 60.355, 68.426, -32.866]
  MoveL 1546 to (-35.13, 161.27, 31.63) mm, rotated rx 180 ry 0 rz 180 deg; joints [-126.078, -65.877, -75.484, 60.355, 68.426, -32.866]
  Call Extruder(395.04040)
  MoveL 1547 to (-35.35, 161.1, 31.63) mm, rotated rx 180 ry 0 rz -180 deg; joints [-126.067, -65.859, -75.536, 60.353, 68.449, -32.838]
  Call Extruder(395.86969)
  MoveL 1548 to (-36.39, 160.19, 31.63) mm, rotated rx 180 ry 0 rz -180 deg; joints [-126.027, -65.766, -75.798, 60.331, 68.554, -32.693]
  Call Extruder(396.50077)
  MoveL 1549 to (-37.09, 159.4, 31.63) mm, rotated rx 180 ry 0 rz 180 deg; joints [-126.014, -65.695, -76.002, 60.298, 68.626, -32.574]
  MoveL 1550 to (-37.09, 159.4, 31.63) mm, rotated rx 180 ry 0 rz 180 deg; joints [-126.014, -65.695, -76.002, 60.298, 68.626, -32.574]
  Call Extruder(396.69836)
  MoveL 1551 to (-37.3, 159.15, 31.63) mm, rotated rx 180 ry 0 rz 180 deg; joints [-126.011, -65.672, -76.066, 60.287, 68.649, -32.537]
  Call Extruder(397.03238)
  MoveL 1552 to (-37.63, 158.7, 31.63) mm, rotated rx -180 ry 0 rz 180 deg; joints [-126.011, -65.634, -76.174, 60.263, 68.684, -32.471]
  MoveL 1553 to (-37.63, 158.7, 31.63) mm, rotated rx -180 ry 0 rz 180 deg; joints [-126.011, -65.634, -76.174, 60.263, 68.684, -32.471]
  Call Extruder(397.26956)
  MoveL 1554 to (-37.87, 158.38, 31.63) mm, rotated rx -180 ry 0 rz 180 deg; joints [-126.011, -65.607, -76.251, 60.246, 68.708, -32.425]
  Set speed (130.0 mm/s)
  MoveL 1555 to (-39.5, 155.42, 31.63) mm, rotated rx 180 ry 0 rz 180 deg; joints [-126.065, -65.381, -76.899, 60.055, 68.889, -32.014]
  MoveL 1556 to (-39.5, 155.42, 41.04) mm, rotated rx -180 ry 0 rz -180 deg; joints [-126.065, -64.048, -77.677, 60.242, 68.613, -32.53]
  Call Extruder(395.26956)
  Set speed (40.0 mm/s)
  MoveL 1557 to (-39.5, 155.42, 41.04) mm, rotated rx -180 ry 0 rz -180 deg; joints [-126.065, -64.048, -77.677, 60.242, 68.613, -32.53]
  Call Extruder(0.00000)
  Set speed (130.0 mm/s)
  MoveL 1558 to (-39.41, 155.44, 41.03) mm, rotated rx 180 ry 0 rz 180 deg; joints [-126.075, -64.053, -77.664, 60.236, 68.604, -32.535]
  Call Extruder(2.00000)
  Set speed (40.0 mm/s)
  MoveL 1559 to (-39.41, 155.44, 41.03) mm, rotated rx 180 ry 0 rz 180 deg; joints [-126.075, -64.053, -77.664, 60.236, 68.604, -32.535]
  Set speed (30.0 mm/s)
  MoveL 1560 to (-39.41, 155.44, 41.03) mm, rotated rx 180 ry 0 rz 180 deg; joints [-126.075, -64.053, -77.664, 60.236, 68.604, -32.535]
  Call Extruder(2.05684)
  MoveL 1561 to (-39.44, 155.34, 41.04) mm, rotated rx 180 ry 0 rz 180 deg; joints [-126.079, -64.047, -77.682, 60.229, 68.607, -32.523]
  MoveL 1562 to (-39.44, 155.34, 41.04) mm, rotated rx 180 ry 0 rz 180 deg; joints [-126.079, -64.047, -77.682, 60.229, 68.607, -32.523]
  Call Extruder(2.17007)
  MoveL 1563 to (-39.5, 155.15, 41.04) mm, rotated rx 180 ry 0 rz -180 deg; joints [-126.087, -64.034, -77.718, 60.213, 68.615, -32.499]
  MoveL 1564 to (-39.5, 155.15, 41.04) mm, rotated rx 180 ry 0 rz -180 deg; joints [-126.087, -64.034, -77.718, 60.213, 68.615, -32.499]
  Call Extruder(2.28286)
  MoveL 1565 to (-39.56, 154.97, 41.04) mm, rotated rx 180 ry 0 rz 180 deg; joints [-126.095, -64.021, -77.754, 60.198, 68.622, -32.474]
  MoveL 1566 to (-39.56, 154.97, 41.04) mm, rotated rx 180 ry 0 rz 180 deg; joints [-126.095, -64.021, -77.754, 60.198, 68.622, -32.474]
  Call Extruder(2.39521)
  MoveL 1567 to (-39.62, 154.78, 41.04) mm, rotated rx -180 ry 0 rz 180 deg; joints [-126.103, -64.008, -77.79, 60.183, 68.629, -32.45]
  MoveL 1568 to (-39.62, 154.78, 41.04) mm, rotated rx -180 ry 0 rz 180 deg; joints [-126.103, -64.008, -77.79, 60.183, 68.629, -32.45]
  Call Extruder(2.50711)
  MoveL 1569 to (-39.68, 154.59, 41.03) mm, rotated rx 180 ry 0 rz 180 deg; joints [-126.111, -63.995, -77.826, 60.167, 68.636, -32.425]
  MoveL 1570 to (-39.68, 154.59, 41.03) mm, rotated rx 180 ry 0 rz 180 deg; joints [-126.111, -63.995, -77.826, 60.167, 68.636, -32.425]
  Call Extruder(2.62851)
  MoveL 1571 to (-39.75, 154.38, 41.03) mm, rotated rx 180 ry 0 rz 180 deg; joints [-126.12, -63.981, -77.866, 60.15, 68.644, -32.399]
  MoveL 1572 to (-39.75, 154.38, 41.03) mm, rotated rx 180 ry 0 rz 180 deg; joints [-126.12, -63.981, -77.866, 60.15, 68.644, -32.399]
  Call Extruder(2.75930)
  MoveL 1573 to (-39.81, 154.16, 41.03) mm, rotated rx 180 ry 0 rz -180 deg; joints [-126.131, -63.966, -77.908, 60.132, 68.652, -32.37]
  MoveL 1574 to (-39.81, 154.16, 41.03) mm, rotated rx 180 ry 0 rz -180 deg; joints [-126.131, -63.966, -77.908, 60.132, 68.652, -32.37]
  Call Extruder(2.88953)
  MoveL 1575 to (-39.88, 153.94, 41.03) mm, rotated rx 180 ry 0 rz 180 deg; joints [-126.141, -63.952, -77.95, 60.113, 68.66, -32.341]
  MoveL 1576 to (-39.88, 153.94, 41.03) mm, rotated rx 180 ry 0 rz 180 deg; joints [-126.141, -63.952, -77.95, 60.113, 68.66, -32.341]
  Call Extruder(3.01920)
  MoveL 1577 to (-39.95, 153.71, 41.04) mm, rotated rx -180 ry 0 rz 180 deg; joints [-126.151, -63.937, -77.993, 60.095, 68.669, -32.312]
  MoveL 1578 to (-39.95, 153.71, 41.04) mm, rotated rx -180 ry 0 rz 180 deg; joints [-126.151, -63.937, -77.993, 60.095, 68.669, -32.312]
  Call Extruder(3.14830)
  MoveL 1579 to (-40.02, 153.49, 41.03) mm, rotated rx -180 ry 0 rz 180 deg; joints [-126.161, -63.922, -78.035, 60.076, 68.677, -32.283]
  MoveL 1580 to (-40.02, 153.49, 41.03) mm, rotated rx -180 ry 0 rz 180 deg; joints [-126.161, -63.922, -78.035, 60.076, 68.677, -32.283]
  Call Extruder(3.26338)
  MoveL 1581 to (-40.06, 153.28, 41.03) mm, rotated rx 180 ry 0 rz -180 deg; joints [-126.173, -63.909, -78.072, 60.058, 68.683, -32.257]
  MoveL 1582 to (-40.06, 153.28, 41.03) mm, rotated rx 180 ry 0 rz -180 deg; joints [-126.173, -63.909, -78.072, 60.058, 68.683, -32.257]
  Call Extruder(3.37802)
  MoveL 1583 to (-40.11, 153.08, 41.04) mm, rotated rx 180 ry 0 rz 180 deg; joints [-126.184, -63.896, -78.108, 60.04, 68.688, -32.232]
  MoveL 1584 to (-40.11, 153.08, 41.04) mm, rotated rx 180 ry 0 rz 180 deg; joints [-126.184, -63.896, -78.108, 60.04, 68.688, -32.232]
  Call Extruder(3.49220)
  MoveL 1585 to (-40.15, 152.88, 41.03) mm, rotated rx 180 ry 0 rz 180 deg; joints [-126.195, -63.883, -78.145, 60.021, 68.694, -32.206]
  MoveL 1586 to (-40.15, 152.88, 41.03) mm, rotated rx 180 ry 0 rz 180 deg; joints [-126.195, -63.883, -78.145, 60.021, 68.694, -32.206]
  Call Extruder(3.60593)
  MoveL 1587 to (-40.2, 152.67, 41.04) mm, rotated rx 180 ry 0 rz 180 deg; joints [-126.206, -63.87, -78.182, 60.003, 68.7, -32.18]
  MoveL 1588 to (-40.2, 152.67, 41.04) mm, rotated rx 180 ry 0 rz 180 deg; joints [-126.206, -63.87, -78.182, 60.003, 68.7, -32.18]
  Call Extruder(3.73136)
  MoveL 1589 to (-40.24, 152.45, 41.04) mm, rotated rx 180 ry 0 rz 180 deg; joints [-126.219, -63.856, -78.222, 59.983, 68.706, -32.152]
  MoveL 1590 to (-40.24, 152.45, 41.04) mm, rotated rx 180 ry 0 rz 180 deg; joints [-126.219, -63.856, -78.222, 59.983, 68.706, -32.152]
  Call Extruder(3.86834)
  MoveL 1591 to (-40.29, 152.2, 41.04) mm, rotated rx -180 ry 0 rz -180 deg; joints [-126.233, -63.84, -78.266, 59.96, 68.713, -32.12]
  MoveL 1592 to (-40.29, 152.2, 41.04) mm, rotated rx -180 ry 0 rz -180 deg; joints [-126.233, -63.84, -78.266, 59.96, 68.713, -32.12]
  Call Extruder(4.00470)
  MoveL 1593 to (-40.34, 151.95, 41.04) mm, rotated rx -180 ry 0 rz 180 deg; joints [-126.248, -63.825, -78.31, 59.938, 68.72, -32.089]
  MoveL 1594 to (-40.34, 151.95, 41.04) mm, rotated rx -180 ry 0 rz 180 deg; joints [-126.248, -63.825, -78.31, 59.938, 68.72, -32.089]
  Call Extruder(4.14046)
  MoveL 1595 to (-40.39, 151.7, 41.04) mm, rotated rx 180 ry 0 rz 180 deg; joints [-126.262, -63.809, -78.354, 59.915, 68.727, -32.058]
  MoveL 1596 to (-40.39, 151.7, 41.04) mm, rotated rx 180 ry 0 rz 180 deg; joints [-126.262, -63.809, -78.354, 59.915, 68.727, -32.058]
  Call Extruder(4.27560)
  MoveL 1597 to (-40.44, 151.45, 41.04) mm, rotated rx -180 ry 0 rz -180 deg; joints [-126.276, -63.794, -78.398, 59.892, 68.733, -32.027]
  MoveL 1598 to (-40.44, 151.45, 41.04) mm, rotated rx -180 ry 0 rz -180 deg; joints [-126.276, -63.794, -78.398, 59.892, 68.733, -32.027]
  Call Extruder(4.41014)
  MoveL 1599 to (-40.49, 151.2, 41.04) mm, rotated rx 180 ry 0 rz 180 deg; joints [-126.291, -63.779, -78.442, 59.87, 68.74, -31.995]
  MoveL 1600 to (-40.49, 151.2, 41.04) mm, rotated rx 180 ry 0 rz 180 deg; joints [-126.291, -63.779, -78.442, 59.87, 68.74, -31.995]
  Call Extruder(4.54406)
  MoveL 1601 to (-40.54, 150.95, 41.04) mm, rotated rx 180 ry 0 rz -180 deg; joints [-126.305, -63.763, -78.486, 59.847, 68.747, -31.964]
  MoveL 1602 to (-40.54, 150.95, 41.04) mm, rotated rx 180 ry 0 rz -180 deg; joints [-126.305, -63.763, -78.486, 59.847, 68.747, -31.964]
  Call Extruder(4.69192)
  MoveL 1603 to (-40.59, 150.67, 41.04) mm, rotated rx -180 ry 0 rz 180 deg; joints [-126.322, -63.746, -78.534, 59.821, 68.753, -31.93]
  MoveL 1604 to (-40.59, 150.67, 41.04) mm, rotated rx -180 ry 0 rz 180 deg; joints [-126.322, -63.746, -78.534, 59.821, 68.753, -31.93]
  Call Extruder(4.85364)
  MoveL 1605 to (-40.64, 150.37, 41.03) mm, rotated rx 180 ry 0 rz -180 deg; joints [-126.341, -63.728, -78.586, 59.793, 68.761, -31.892]
  MoveL 1606 to (-40.64, 150.37, 41.03) mm, rotated rx 180 ry 0 rz -180 deg; joints [-126.341, -63.728, -78.586, 59.793, 68.761, -31.892]
  Call Extruder(5.01464)
  MoveL 1607 to (-40.69, 150.06, 41.03) mm, rotated rx -180 ry 0 rz 180 deg; joints [-126.36, -63.71, -78.639, 59.764, 68.768, -31.854]
  MoveL 1608 to (-40.69, 150.06, 41.03) mm, rotated rx -180 ry 0 rz 180 deg; joints [-126.36, -63.71, -78.639, 59.764, 68.768, -31.854]
  Call Extruder(5.17491)
  MoveL 1609 to (-40.74, 149.76, 41.03) mm, rotated rx -180 ry 0 rz 180 deg; joints [-126.379, -63.691, -78.691, 59.735, 68.775, -31.816]
  MoveL 1610 to (-40.74, 149.76, 41.03) mm, rotated rx -180 ry 0 rz 180 deg; joints [-126.379, -63.691, -78.691, 59.735, 68.775, -31.816]
  Call Extruder(5.33445)
  MoveL 1611 to (-40.78, 149.45, 41.03) mm, rotated rx -180 ry 0 rz 180 deg; joints [-126.398, -63.673, -78.743, 59.706, 68.782, -31.778]
  MoveL 1612 to (-40.78, 149.45, 41.03) mm, rotated rx -180 ry 0 rz 180 deg; joints [-126.398, -63.673, -78.743, 59.706, 68.782, -31.778]
  Call Extruder(5.49326)
  MoveL 1613 to (-40.83, 149.14, 41.04) mm, rotated rx -180 ry 0 rz 180 deg; joints [-126.417, -63.655, -78.796, 59.678, 68.789, -31.741]
  MoveL 1614 to (-40.83, 149.14, 41.04) mm, rotated rx -180 ry 0 rz 180 deg; joints [-126.417, -63.655, -78.796, 59.678, 68.789, -31.741]
  Call Extruder(5.67193)
  MoveL 1615 to (-40.88, 148.8, 41.03) mm, rotated rx -180 ry 0 rz 180 deg; joints [-126.439, -63.634, -78.854, 59.644, 68.796, -31.698]
  MoveL 1616 to (-40.88, 148.8, 41.03) mm, rotated rx -180 ry 0 rz 180 deg; joints [-126.439, -63.634, -78.854, 59.644, 68.796, -31.698]
  Call Extruder(5.87037)
  MoveL 1617 to (-40.92, 148.41, 41.04) mm, rotated rx 180 ry 0 rz 180 deg; joints [-126.465, -63.612, -78.918, 59.607, 68.804, -31.651]
  MoveL 1618 to (-40.92, 148.41, 41.04) mm, rotated rx 180 ry 0 rz 180 deg; joints [-126.465, -63.612, -78.918, 59.607, 68.804, -31.651]
  Call Extruder(6.06794)
  MoveL 1619 to (-40.97, 148.02, 41.04) mm, rotated rx 180 ry 0 rz 180 deg; joints [-126.491, -63.589, -78.983, 59.569, 68.812, -31.603]
  MoveL 1620 to (-40.97, 148.02, 41.04) mm, rotated rx 180 ry 0 rz 180 deg; joints [-126.491, -63.589, -78.983, 59.569, 68.812, -31.603]
  Call Extruder(6.26465)
  MoveL 1621 to (-41.02, 147.63, 41.03) mm, rotated rx 180 ry 0 rz -180 deg; joints [-126.517, -63.567, -79.047, 59.531, 68.819, -31.556]
  MoveL 1622 to (-41.02, 147.63, 41.03) mm, rotated rx 180 ry 0 rz -180 deg; joints [-126.517, -63.567, -79.047, 59.531, 68.819, -31.556]
  Call Extruder(6.46049)
  MoveL 1623 to (-41.06, 147.25, 41.04) mm, rotated rx 180 ry 0 rz 180 deg; joints [-126.543, -63.545, -79.111, 59.493, 68.827, -31.509]
  MoveL 1624 to (-41.06, 147.25, 41.04) mm, rotated rx 180 ry 0 rz 180 deg; joints [-126.543, -63.545, -79.111, 59.493, 68.827, -31.509]
  Call Extruder(6.75588)
  MoveL 1625 to (-41.11, 146.66, 41.04) mm, rotated rx -180 ry 0 rz 180 deg; joints [-126.585, -63.512, -79.206, 59.434, 68.836, -31.437]
  MoveL 1626 to (-41.11, 146.66, 41.04) mm, rotated rx -180 ry 0 rz 180 deg; joints [-126.585, -63.512, -79.206, 59.434, 68.836, -31.437]
  Call Extruder(7.04995)
  MoveL 1627 to (-41.15, 146.07, 41.04) mm, rotated rx 180 ry 0 rz 180 deg; joints [-126.628, -63.479, -79.301, 59.375, 68.846, -31.366]
  MoveL 1628 to (-41.15, 146.07, 41.04) mm, rotated rx 180 ry 0 rz 180 deg; joints [-126.628, -63.479, -79.301, 59.375, 68.846, -31.366]
  Call Extruder(7.34268)
  MoveL 1629 to (-41.2, 145.48, 41.03) mm, rotated rx -180 ry 0 rz -180 deg; joints [-126.67, -63.446, -79.396, 59.315, 68.855, -31.295]
  MoveL 1630 to (-41.2, 145.48, 41.03) mm, rotated rx -180 ry 0 rz -180 deg; joints [-126.67, -63.446, -79.396, 59.315, 68.855, -31.295]
  Call Extruder(7.91614)
  MoveL 1631 to (-41.25, 144.32, 41.04) mm, rotated rx 180 ry 0 rz 180 deg; joints [-126.759, -63.383, -79.577, 59.194, 68.87, -31.157]
  MoveL 1632 to (-41.25, 144.32, 41.04) mm, rotated rx 180 ry 0 rz 180 deg; joints [-126.759, -63.383, -79.577, 59.194, 68.87, -31.157]
  Call Extruder(8.63010)
  MoveL 1633 to (-41.29, 142.86, 41.03) mm, rotated rx -180 ry 0 rz 180 deg; joints [-126.873, -63.306, -79.801, 59.041, 68.886, -30.984]
  Call Extruder(50.69492)
  MoveL 1634 to (-41.29, 57.14, 41.03) mm, rotated rx 180 ry 0 rz 180 deg; joints [-135.148, -59.724, -91.342, 48.662, 69.941, -21.3]
  Call Extruder(51.12347)
  MoveL 1635 to (-41.27, 56.26, 41.04) mm, rotated rx 180 ry 0 rz -180 deg; joints [-135.25, -59.696, -91.443, 48.541, 69.953, -21.207]
  MoveL 1636 to (-41.27, 56.26, 41.04) mm, rotated rx 180 ry 0 rz -180 deg; joints [-135.25, -59.696, -91.443, 48.541, 69.953, -21.207]
  Call Extruder(51.69692)
  MoveL 1637 to (-41.23, 55.1, 41.03) mm, rotated rx 180 ry 0 rz 180 deg; joints [-135.387, -59.661, -91.575, 48.377, 69.967, -21.083]
  MoveL 1638 to (-41.23, 55.1, 41.03) mm, rotated rx 180 ry 0 rz 180 deg; joints [-135.387, -59.661, -91.575, 48.377, 69.967, -21.083]
  Call Extruder(52.13124)
  MoveL 1639 to (-41.18, 54.23, 41.04) mm, rotated rx 180 ry 0 rz 180 deg; joints [-135.493, -59.634, -91.673, 48.253, 69.977, -20.99]
  MoveL 1640 to (-41.18, 54.23, 41.04) mm, rotated rx 180 ry 0 rz 180 deg; joints [-135.493, -59.634, -91.673, 48.253, 69.977, -20.99]
  Call Extruder(52.42530)
  MoveL 1641 to (-41.13, 53.64, 41.04) mm, rotated rx 180 ry 0 rz 180 deg; joints [-135.566, -59.617, -91.737, 48.167, 69.982, -20.928]
  MoveL 1642 to (-41.13, 53.64, 41.04) mm, rotated rx 180 ry 0 rz 180 deg; joints [-135.566, -59.617, -91.737, 48.167, 69.982, -20.928]
  Call Extruder(52.72070)
  MoveL 1643 to (-41.09, 53.05, 41.04) mm, rotated rx 180 ry 0 rz 180 deg; joints [-135.64, -59.6, -91.801, 48.082, 69.987, -20.866]
  MoveL 1644 to (-41.09, 53.05, 41.04) mm, rotated rx 180 ry 0 rz 180 deg; joints [-135.64, -59.6, -91.801, 48.082, 69.987, -20.866]
  Call Extruder(52.96694)
  MoveL 1645 to (-41.04, 52.56, 41.03) mm, rotated rx -180 ry 0 rz 180 deg; joints [-135.701, -59.586, -91.852, 48.011, 69.99, -20.815]
  MoveL 1646 to (-41.04, 52.56, 41.03) mm, rotated rx -180 ry 0 rz 180 deg; joints [-135.701, -59.586, -91.852, 48.011, 69.99, -20.815]
  Call Extruder(53.16365)
  MoveL 1647 to (-40.99, 52.17, 41.04) mm, rotated rx 180 ry 0 rz 180 deg; joints [-135.751, -59.576, -91.892, 47.953, 69.992, -20.775]
  MoveL 1648 to (-40.99, 52.17, 41.04) mm, rotated rx 180 ry 0 rz 180 deg; joints [-135.751, -59.576, -91.892, 47.953, 69.992, -20.775]
  Call Extruder(53.36122)
  MoveL 1649 to (-40.95, 51.78, 41.04) mm, rotated rx 180 ry 0 rz 180 deg; joints [-135.801, -59.565, -91.932, 47.895, 69.994, -20.735]
  MoveL 1650 to (-40.95, 51.78, 41.04) mm, rotated rx 180 ry 0 rz 180 deg; joints [-135.801, -59.565, -91.932, 47.895, 69.994, -20.735]
  Call Extruder(53.55966)
  MoveL 1651 to (-40.9, 51.4, 41.04) mm, rotated rx 180 ry 0 rz -180 deg; joints [-135.852, -59.555, -91.972, 47.837, 69.996, -20.695]
  MoveL 1652 to (-40.9, 51.4, 41.04) mm, rotated rx 180 ry 0 rz -180 deg; joints [-135.852, -59.555, -91.972, 47.837, 69.996, -20.695]
  Call Extruder(53.75897)
  MoveL 1653 to (-40.86, 51.01, 41.04) mm, rotated rx 180 ry 0 rz 180 deg; joints [-135.902, -59.544, -92.011, 47.779, 69.997, -20.655]
  MoveL 1654 to (-40.86, 51.01, 41.04) mm, rotated rx 180 ry 0 rz 180 deg; joints [-135.902, -59.544, -92.011, 47.779, 69.997, -20.655]
  Call Extruder(53.91779)
  MoveL 1655 to (-40.81, 50.7, 41.04) mm, rotated rx 180 ry 0 rz -180 deg; joints [-135.943, -59.536, -92.041, 47.733, 69.998, -20.624]
  MoveL 1656 to (-40.81, 50.7, 41.04) mm, rotated rx 180 ry 0 rz -180 deg; joints [-135.943, -59.536, -92.041, 47.733, 69.998, -20.624]
  Call Extruder(54.07733)
  MoveL 1657 to (-40.76, 50.4, 41.03) mm, rotated rx 180 ry 0 rz -180 deg; joints [-135.984, -59.528, -92.071, 47.686, 69.998, -20.592]
  MoveL 1658 to (-40.76, 50.4, 41.03) mm, rotated rx 180 ry 0 rz -180 deg; joints [-135.984, -59.528, -92.071, 47.686, 69.998, -20.592]
  Call Extruder(54.23760)
  MoveL 1659 to (-40.71, 50.09, 41.04) mm, rotated rx -180 ry 0 rz 180 deg; joints [-136.025, -59.52, -92.1, 47.639, 69.998, -20.561]
  MoveL 1660 to (-40.71, 50.09, 41.04) mm, rotated rx -180 ry 0 rz 180 deg; joints [-136.025, -59.52, -92.1, 47.639, 69.998, -20.561]
  Call Extruder(54.39860)
  MoveL 1661 to (-40.66, 49.79, 41.03) mm, rotated rx -180 ry 0 rz -180 deg; joints [-136.067, -59.512, -92.13, 47.592, 69.998, -20.53]
  MoveL 1662 to (-40.66, 49.79, 41.03) mm, rotated rx -180 ry 0 rz -180 deg; joints [-136.067, -59.512, -92.13, 47.592, 69.998, -20.53]
  Call Extruder(54.56032)
  MoveL 1663 to (-40.61, 49.48, 41.04) mm, rotated rx -180 ry 0 rz 180 deg; joints [-136.108, -59.505, -92.16, 47.545, 69.999, -20.499]
  MoveL 1664 to (-40.61, 49.48, 41.04) mm, rotated rx -180 ry 0 rz 180 deg; joints [-136.108, -59.505, -92.16, 47.545, 69.999, -20.499]
  Call Extruder(54.72278)
  MoveL 1665 to (-40.56, 49.18, 41.04) mm, rotated rx 180 ry 0 rz -180 deg; joints [-136.149, -59.497, -92.189, 47.498, 69.999, -20.468]
  MoveL 1666 to (-40.56, 49.18, 41.04) mm, rotated rx 180 ry 0 rz -180 deg; joints [-136.149, -59.497, -92.189, 47.498, 69.999, -20.468]
  Call Extruder(54.85670)
  MoveL 1667 to (-40.52, 48.93, 41.04) mm, rotated rx 180 ry 0 rz 180 deg; joints [-136.184, -59.491, -92.212, 47.459, 69.998, -20.443]
  MoveL 1668 to (-40.52, 48.93, 41.04) mm, rotated rx 180 ry 0 rz 180 deg; joints [-136.184, -59.491, -92.212, 47.459, 69.998, -20.443]
  Call Extruder(54.99124)
  MoveL 1669 to (-40.47, 48.68, 41.03) mm, rotated rx -180 ry 0 rz 180 deg; joints [-136.219, -59.485, -92.235, 47.419, 69.997, -20.418]
  MoveL 1670 to (-40.47, 48.68, 41.03) mm, rotated rx -180 ry 0 rz 180 deg; joints [-136.219, -59.485, -92.235, 47.419, 69.997, -20.418]
  Call Extruder(55.12638)
  MoveL 1671 to (-40.42, 48.43, 41.03) mm, rotated rx -180 ry 0 rz -180 deg; joints [-136.254, -59.479, -92.258, 47.38, 69.996, -20.393]
  MoveL 1672 to (-40.42, 48.43, 41.03) mm, rotated rx -180 ry 0 rz -180 deg; joints [-136.254, -59.479, -92.258, 47.38, 69.996, -20.393]
  Call Extruder(55.26214)
  MoveL 1673 to (-40.37, 48.18, 41.03) mm, rotated rx 180 ry 0 rz 180 deg; joints [-136.288, -59.473, -92.281, 47.341, 69.996, -20.367]
  MoveL 1674 to (-40.37, 48.18, 41.03) mm, rotated rx 180 ry 0 rz 180 deg; joints [-136.288, -59.473, -92.281, 47.341, 69.996, -20.367]
  Call Extruder(55.39850)
  MoveL 1675 to (-40.32, 47.93, 41.04) mm, rotated rx 180 ry 0 rz 180 deg; joints [-136.323, -59.467, -92.303, 47.301, 69.995, -20.342]
  MoveL 1676 to (-40.32, 47.93, 41.04) mm, rotated rx 180 ry 0 rz 180 deg; joints [-136.323, -59.467, -92.303, 47.301, 69.995, -20.342]
  Call Extruder(55.53548)
  MoveL 1677 to (-40.27, 47.68, 41.04) mm, rotated rx -180 ry 0 rz 180 deg; joints [-136.358, -59.461, -92.326, 47.262, 69.994, -20.317]
  MoveL 1678 to (-40.27, 47.68, 41.04) mm, rotated rx -180 ry 0 rz 180 deg; joints [-136.358, -59.461, -92.326, 47.262, 69.994, -20.317]
  Call Extruder(55.67306)
  MoveL 1679 to (-40.22, 47.43, 41.04) mm, rotated rx 180 ry 0 rz 180 deg; joints [-136.393, -59.455, -92.349, 47.223, 69.993, -20.292]
  MoveL 1680 to (-40.22, 47.43, 41.04) mm, rotated rx 180 ry 0 rz 180 deg; joints [-136.393, -59.455, -92.349, 47.223, 69.993, -20.292]
  Call Extruder(55.78679)
  MoveL 1681 to (-40.17, 47.23, 41.04) mm, rotated rx 180 ry 0 rz -180 deg; joints [-136.422, -59.45, -92.367, 47.19, 69.992, -20.272]
  MoveL 1682 to (-40.17, 47.23, 41.04) mm, rotated rx 180 ry 0 rz -180 deg; joints [-136.422, -59.45, -92.367, 47.19, 69.992, -20.272]
  Call Extruder(55.90097)
  MoveL 1683 to (-40.13, 47.02, 41.03) mm, rotated rx -180 ry 0 rz 180 deg; joints [-136.452, -59.445, -92.385, 47.157, 69.991, -20.252]
  MoveL 1684 to (-40.13, 47.02, 41.03) mm, rotated rx -180 ry 0 rz 180 deg; joints [-136.452, -59.445, -92.385, 47.157, 69.991, -20.252]
  Call Extruder(56.01561)
  MoveL 1685 to (-40.08, 46.82, 41.04) mm, rotated rx 180 ry 0 rz -180 deg; joints [-136.481, -59.441, -92.403, 47.125, 69.99, -20.231]
  MoveL 1686 to (-40.08, 46.82, 41.04) mm, rotated rx 180 ry 0 rz -180 deg; joints [-136.481, -59.441, -92.403, 47.125, 69.99, -20.231]
  Call Extruder(56.13069)
  MoveL 1687 to (-40.04, 46.61, 41.04) mm, rotated rx -180 ry 0 rz -180 deg; joints [-136.51, -59.436, -92.421, 47.092, 69.989, -20.211]
  MoveL 1688 to (-40.04, 46.61, 41.04) mm, rotated rx -180 ry 0 rz -180 deg; joints [-136.51, -59.436, -92.421, 47.092, 69.989, -20.211]
  Call Extruder(56.25293)
  MoveL 1689 to (-39.98, 46.4, 41.04) mm, rotated rx 180 ry 0 rz -180 deg; joints [-136.542, -59.431, -92.439, 47.057, 69.987, -20.19]
  MoveL 1690 to (-39.98, 46.4, 41.04) mm, rotated rx 180 ry 0 rz -180 deg; joints [-136.542, -59.431, -92.439, 47.057, 69.987, -20.19]
  Call Extruder(56.38259)
  MoveL 1691 to (-39.92, 46.18, 41.04) mm, rotated rx 180 ry 0 rz 180 deg; joints [-136.576, -59.427, -92.456, 47.019, 69.984, -20.168]
  MoveL 1692 to (-39.92, 46.18, 41.04) mm, rotated rx 180 ry 0 rz 180 deg; joints [-136.576, -59.427, -92.456, 47.019, 69.984, -20.168]
  Call Extruder(56.51282)
  MoveL 1693 to (-39.85, 45.95, 41.04) mm, rotated rx 180 ry 0 rz 180 deg; joints [-136.61, -59.422, -92.474, 46.982, 69.981, -20.147]
  MoveL 1694 to (-39.85, 45.95, 41.04) mm, rotated rx 180 ry 0 rz 180 deg; joints [-136.61, -59.422, -92.474, 46.982, 69.981, -20.147]
  Call Extruder(56.64361)
  MoveL 1695 to (-39.78, 45.73, 41.04) mm, rotated rx 180 ry 0 rz 180 deg; joints [-136.644, -59.417, -92.491, 46.944, 69.978, -20.125]
  MoveL 1696 to (-39.78, 45.73, 41.04) mm, rotated rx 180 ry 0 rz 180 deg; joints [-136.644, -59.417, -92.491, 46.944, 69.978, -20.125]
  Call Extruder(56.77497)
  MoveL 1697 to (-39.71, 45.51, 41.04) mm, rotated rx 180 ry 0 rz 180 deg; joints [-136.678, -59.413, -92.509, 46.907, 69.975, -20.103]
  MoveL 1698 to (-39.71, 45.51, 41.04) mm, rotated rx 180 ry 0 rz 180 deg; joints [-136.678, -59.413, -92.509, 46.907, 69.975, -20.103]
  Call Extruder(56.88687)
  MoveL 1699 to (-39.65, 45.32, 41.04) mm, rotated rx 180 ry 0 rz -180 deg; joints [-136.707, -59.409, -92.523, 46.875, 69.972, -20.085]
  MoveL 1700 to (-39.65, 45.32, 41.04) mm, rotated rx 180 ry 0 rz -180 deg; joints [-136.707, -59.409, -92.523, 46.875, 69.972, -20.085]
  Call Extruder(56.99922)
  MoveL 1701 to (-39.59, 45.13, 41.03) mm, rotated rx -180 ry 0 rz 180 deg; joints [-136.737, -59.406, -92.537, 46.843, 69.969, -20.067]
  MoveL 1702 to (-39.59, 45.13, 41.03) mm, rotated rx -180 ry 0 rz 180 deg; joints [-136.737, -59.406, -92.537, 46.843, 69.969, -20.067]
  Call Extruder(57.11201)
  MoveL 1703 to (-39.53, 44.94, 41.04) mm, rotated rx -180 ry 0 rz 180 deg; joints [-136.766, -59.402, -92.551, 46.81, 69.966, -20.049]
  MoveL 1704 to (-39.53, 44.94, 41.04) mm, rotated rx -180 ry 0 rz 180 deg; joints [-136.766, -59.402, -92.551, 46.81, 69.966, -20.049]
  Call Extruder(57.22525)
  MoveL 1705 to (-39.47, 44.75, 41.04) mm, rotated rx 180 ry 0 rz -180 deg; joints [-136.796, -59.398, -92.565, 46.778, 69.963, -20.031]
  MoveL 1706 to (-39.47, 44.75, 41.04) mm, rotated rx 180 ry 0 rz -180 deg; joints [-136.796, -59.398, -92.565, 46.778, 69.963, -20.031]
  Call Extruder(57.33893)
  MoveL 1707 to (-39.41, 44.56, 41.04) mm, rotated rx 180 ry 0 rz 180 deg; joints [-136.825, -59.395, -92.579, 46.746, 69.961, -20.013]
  MoveL 1708 to (-39.41, 44.56, 41.04) mm, rotated rx 180 ry 0 rz 180 deg; joints [-136.825, -59.395, -92.579, 46.746, 69.961, -20.013]
  Call Extruder(57.52088)
  MoveL 1709 to (-39.29, 44.27, 41.04) mm, rotated rx 180 ry 0 rz -180 deg; joints [-136.873, -59.39, -92.598, 46.694, 69.953, -19.985]
  MoveL 1710 to (-39.29, 44.27, 41.04) mm, rotated rx 180 ry 0 rz -180 deg; joints [-136.873, -59.39, -92.598, 46.694, 69.953, -19.985]
  Call Extruder(57.70360)
  MoveL 1711 to (-39.16, 43.98, 41.04) mm, rotated rx 180 ry 0 rz -180 deg; joints [-136.922, -59.385, -92.616, 46.642, 69.946, -19.958]
  MoveL 1712 to (-39.16, 43.98, 41.04) mm, rotated rx 180 ry 0 rz -180 deg; joints [-136.922, -59.385, -92.616, 46.642, 69.946, -19.958]
  Call Extruder(57.87401)
  MoveL 1713 to (-39.05, 43.71, 41.03) mm, rotated rx 180 ry 0 rz 180 deg; joints [-136.967, -59.381, -92.633, 46.594, 69.939, -19.933]
  MoveL 1714 to (-39.05, 43.71, 41.03) mm, rotated rx 180 ry 0 rz 180 deg; joints [-136.967, -59.381, -92.633, 46.594, 69.939, -19.933]
  Call Extruder(58.03200)
  MoveL 1715 to (-38.94, 43.46, 41.03) mm, rotated rx 180 ry 0 rz 180 deg; joints [-137.009, -59.377, -92.648, 46.549, 69.933, -19.91]
  MoveL 1716 to (-38.94, 43.46, 41.03) mm, rotated rx 180 ry 0 rz 180 deg; joints [-137.009, -59.377, -92.648, 46.549, 69.933, -19.91]
  Call Extruder(58.19059)
  MoveL 1717 to (-38.84, 43.21, 41.04) mm, rotated rx 180 ry 0 rz 180 deg; joints [-137.05, -59.373, -92.663, 46.504, 69.926, -19.887]
  MoveL 1718 to (-38.84, 43.21, 41.04) mm, rotated rx 180 ry 0 rz 180 deg; joints [-137.05, -59.373, -92.663, 46.504, 69.926, -19.887]
  Call Extruder(58.39676)
  MoveL 1719 to (-38.66, 42.91, 41.04) mm, rotated rx 180 ry 0 rz -180 deg; joints [-137.107, -59.369, -92.677, 46.445, 69.914, -19.86]
  MoveL 1720 to (-38.66, 42.91, 41.04) mm, rotated rx 180 ry 0 rz -180 deg; joints [-137.107, -59.369, -92.677, 46.445, 69.914, -19.86]
  Call Extruder(58.60370)
  MoveL 1721 to (-38.49, 42.6, 41.04) mm, rotated rx 180 ry 0 rz -180 deg; joints [-137.163, -59.366, -92.69, 46.386, 69.902, -19.833]
  MoveL 1722 to (-38.49, 42.6, 41.04) mm, rotated rx 180 ry 0 rz -180 deg; joints [-137.163, -59.366, -92.69, 46.386, 69.902, -19.833]
  Call Extruder(58.81142)
  MoveL 1723 to (-38.31, 42.3, 41.04) mm, rotated rx 180 ry 0 rz 180 deg; joints [-137.219, -59.362, -92.703, 46.328, 69.889, -19.807]
  MoveL 1724 to (-38.31, 42.3, 41.04) mm, rotated rx 180 ry 0 rz 180 deg; joints [-137.219, -59.362, -92.703, 46.328, 69.889, -19.807]
  Call Extruder(59.01993)
  MoveL 1725 to (-38.13, 41.99, 41.04) mm, rotated rx 180 ry 0 rz 180 deg; joints [-137.275, -59.359, -92.715, 46.269, 69.877, -19.78]
  MoveL 1726 to (-38.13, 41.99, 41.04) mm, rotated rx 180 ry 0 rz 180 deg; joints [-137.275, -59.359, -92.715, 46.269, 69.877, -19.78]
  Call Extruder(59.19948)
  MoveL 1727 to (-37.96, 41.75, 41.03) mm, rotated rx 180 ry 0 rz 180 deg; joints [-137.324, -59.357, -92.721, 46.218, 69.863, -19.759]
  MoveL 1728 to (-37.96, 41.75, 41.03) mm, rotated rx 180 ry 0 rz 180 deg; joints [-137.324, -59.357, -92.721, 46.218, 69.863, -19.759]
  Call Extruder(59.53291)
  MoveL 1729 to (-37.63, 41.3, 41.03) mm, rotated rx 180 ry 0 rz 180 deg; joints [-137.415, -59.355, -92.732, 46.125, 69.838, -19.722]
  MoveL 1730 to (-37.63, 41.3, 41.03) mm, rotated rx 180 ry 0 rz 180 deg; joints [-137.415, -59.355, -92.732, 46.125, 69.838, -19.722]
  Call Extruder(59.86753)
  MoveL 1731 to (-37.3, 40.85, 41.03) mm, rotated rx 180 ry 0 rz -180 deg; joints [-137.506, -59.352, -92.743, 46.032, 69.813, -19.684]
  Call Extruder(60.69546)
  MoveL 1732 to (-36.39, 39.81, 41.03) mm, rotated rx -180 ry 0 rz -180 deg; joints [-137.733, -59.351, -92.747, 45.803, 69.739, -19.603]
  Call Extruder(61.52337)
  MoveL 1733 to (-35.35, 38.9, 41.03) mm, rotated rx -180 ry 0 rz -180 deg; joints [-137.958, -59.358, -92.721, 45.582, 69.65, -19.54]
  Call Extruder(61.69068)
  MoveL 1734 to (-35.13, 38.73, 41.03) mm, rotated rx -180 ry 0 rz -180 deg; joints [-138.003, -59.36, -92.711, 45.539, 69.63, -19.529]
  MoveL 1735 to (-35.13, 38.73, 41.03) mm, rotated rx -180 ry 0 rz -180 deg; joints [-138.003, -59.36, -92.711, 45.539, 69.63, -19.529]
  Call Extruder(62.02410)
  MoveL 1736 to (-34.68, 38.4, 41.03) mm, rotated rx -180 ry 0 rz 180 deg; joints [-138.092, -59.365, -92.692, 45.453, 69.59, -19.509]
  MoveL 1737 to (-34.68, 38.4, 41.03) mm, rotated rx -180 ry 0 rz 180 deg; joints [-138.092, -59.365, -92.692, 45.453, 69.59, -19.509]
  Call Extruder(62.35635)
  MoveL 1738 to (-34.23, 38.08, 41.04) mm, rotated rx 180 ry 0 rz -180 deg; joints [-138.182, -59.37, -92.672, 45.367, 69.55, -19.488]
  MoveL 1739 to (-34.23, 38.08, 41.04) mm, rotated rx 180 ry 0 rz -180 deg; joints [-138.182, -59.37, -92.672, 45.367, 69.55, -19.488]
  Call Extruder(62.47405)
  MoveL 1740 to (-34.05, 37.98, 41.04) mm, rotated rx 180 ry 0 rz 180 deg; joints [-138.213, -59.373, -92.662, 45.338, 69.534, -19.483]
  MoveL 1741 to (-34.05, 37.98, 41.04) mm, rotated rx 180 ry 0 rz 180 deg; joints [-138.213, -59.373, -92.662, 45.338, 69.534, -19.483]
  Call Extruder(62.68177)
  MoveL 1742 to (-33.75, 37.8, 41.03) mm, rotated rx -180 ry 0 rz 180 deg; joints [-138.267, -59.378, -92.644, 45.286, 69.507, -19.474]
  MoveL 1743 to (-33.75, 37.8, 41.03) mm, rotated rx -180 ry 0 rz 180 deg; joints [-138.267, -59.378, -92.644, 45.286, 69.507, -19.474]
  Call Extruder(62.88871)
  MoveL 1744 to (-33.45, 37.63, 41.03) mm, rotated rx 180 ry 0 rz -180 deg; joints [-138.322, -59.382, -92.626, 45.235, 69.479, -19.465]
  MoveL 1745 to (-33.45, 37.63, 41.03) mm, rotated rx 180 ry 0 rz -180 deg; joints [-138.322, -59.382, -92.626, 45.235, 69.479, -19.465]
  Call Extruder(63.09487)
  MoveL 1746 to (-33.14, 37.45, 41.04) mm, rotated rx 180 ry 0 rz 180 deg; joints [-138.376, -59.387, -92.607, 45.184, 69.451, -19.456]
  MoveL 1747 to (-33.14, 37.45, 41.04) mm, rotated rx 180 ry 0 rz 180 deg; joints [-138.376, -59.387, -92.607, 45.184, 69.451, -19.456]
  Call Extruder(63.27655)
  MoveL 1748 to (-32.87, 37.31, 41.03) mm, rotated rx -180 ry 0 rz 180 deg; joints [-138.424, -59.392, -92.588, 45.139, 69.425, -19.45]
  MoveL 1749 to (-32.87, 37.31, 41.03) mm, rotated rx -180 ry 0 rz 180 deg; joints [-138.424, -59.392, -92.588, 45.139, 69.425, -19.45]
  Call Extruder(63.43455)
  MoveL 1750 to (-32.62, 37.2, 41.04) mm, rotated rx 180 ry 0 rz -180 deg; joints [-138.464, -59.397, -92.569, 45.103, 69.402, -19.447]
  MoveL 1751 to (-32.62, 37.2, 41.04) mm, rotated rx 180 ry 0 rz -180 deg; joints [-138.464, -59.397, -92.569, 45.103, 69.402, -19.447]
  Call Extruder(63.59195)
  MoveL 1752 to (-32.37, 37.1, 41.04) mm, rotated rx 180 ry 0 rz 180 deg; joints [-138.504, -59.402, -92.55, 45.066, 69.379, -19.443]
  MoveL 1753 to (-32.37, 37.1, 41.04) mm, rotated rx 180 ry 0 rz 180 deg; joints [-138.504, -59.402, -92.55, 45.066, 69.379, -19.443]
  Call Extruder(63.77466)
  MoveL 1754 to (-32.07, 36.98, 41.04) mm, rotated rx 180 ry 0 rz -180 deg; joints [-138.551, -59.408, -92.527, 45.024, 69.351, -19.44]
  MoveL 1755 to (-32.07, 36.98, 41.04) mm, rotated rx 180 ry 0 rz -180 deg; joints [-138.551, -59.408, -92.527, 45.024, 69.351, -19.44]
  Call Extruder(63.95661)
  MoveL 1756 to (-31.78, 36.85, 41.04) mm, rotated rx 180 ry 0 rz -180 deg; joints [-138.597, -59.414, -92.504, 44.982, 69.324, -19.436]
  MoveL 1757 to (-31.78, 36.85, 41.04) mm, rotated rx 180 ry 0 rz -180 deg; joints [-138.597, -59.414, -92.504, 44.982, 69.324, -19.436]
  Call Extruder(64.10394)
  MoveL 1758 to (-31.54, 36.76, 41.03) mm, rotated rx 180 ry 0 rz 180 deg; joints [-138.634, -59.419, -92.484, 44.948, 69.301, -19.434]
  MoveL 1759 to (-31.54, 36.76, 41.03) mm, rotated rx 180 ry 0 rz 180 deg; joints [-138.634, -59.419, -92.484, 44.948, 69.301, -19.434]
  Call Extruder(64.21718)
  MoveL 1760 to (-31.35, 36.7, 41.04) mm, rotated rx 180 ry 0 rz -180 deg; joints [-138.662, -59.424, -92.467, 44.923, 69.283, -19.433]
  MoveL 1761 to (-31.35, 36.7, 41.04) mm, rotated rx 180 ry 0 rz -180 deg; joints [-138.662, -59.424, -92.467, 44.923, 69.283, -19.433]
  Call Extruder(64.32997)
  MoveL 1762 to (-31.17, 36.64, 41.04) mm, rotated rx 180 ry 0 rz 180 deg; joints [-138.69, -59.428, -92.45, 44.899, 69.265, -19.433]
  MoveL 1763 to (-31.17, 36.64, 41.04) mm, rotated rx 180 ry 0 rz 180 deg; joints [-138.69, -59.428, -92.45, 44.899, 69.265, -19.433]
  Call Extruder(64.44232)
  MoveL 1764 to (-30.98, 36.58, 41.04) mm, rotated rx -180 ry 0 rz 180 deg; joints [-138.718, -59.433, -92.433, 44.874, 69.247, -19.432]
  MoveL 1765 to (-30.98, 36.58, 41.04) mm, rotated rx -180 ry 0 rz 180 deg; joints [-138.718, -59.433, -92.433, 44.874, 69.247, -19.432]
  Call Extruder(64.55422)
  MoveL 1766 to (-30.79, 36.52, 41.04) mm, rotated rx -180 ry 0 rz 180 deg; joints [-138.745, -59.437, -92.416, 44.849, 69.228, -19.432]
  MoveL 1767 to (-30.79, 36.52, 41.04) mm, rotated rx -180 ry 0 rz 180 deg; joints [-138.745, -59.437, -92.416, 44.849, 69.228, -19.432]
  Call Extruder(64.67562)
  MoveL 1768 to (-30.58, 36.45, 41.04) mm, rotated rx 180 ry 0 rz -180 deg; joints [-138.776, -59.442, -92.397, 44.823, 69.209, -19.432]
  MoveL 1769 to (-30.58, 36.45, 41.04) mm, rotated rx 180 ry 0 rz -180 deg; joints [-138.776, -59.442, -92.397, 44.823, 69.209, -19.432]
  Call Extruder(64.80641)
  MoveL 1770 to (-30.36, 36.39, 41.04) mm, rotated rx 180 ry 0 rz -180 deg; joints [-138.808, -59.447, -92.377, 44.794, 69.187, -19.431]
  MoveL 1771 to (-30.36, 36.39, 41.04) mm, rotated rx 180 ry 0 rz -180 deg; joints [-138.808, -59.447, -92.377, 44.794, 69.187, -19.431]
  Call Extruder(64.93664)
  MoveL 1772 to (-30.14, 36.32, 41.03) mm, rotated rx -180 ry 0 rz 180 deg; joints [-138.84, -59.453, -92.356, 44.766, 69.166, -19.431]
  MoveL 1773 to (-30.14, 36.32, 41.03) mm, rotated rx -180 ry 0 rz 180 deg; joints [-138.84, -59.453, -92.356, 44.766, 69.166, -19.431]
  Call Extruder(65.06630)
  MoveL 1774 to (-29.91, 36.25, 41.04) mm, rotated rx 180 ry 0 rz -180 deg; joints [-138.873, -59.458, -92.335, 44.737, 69.144, -19.431]
  MoveL 1775 to (-29.91, 36.25, 41.04) mm, rotated rx 180 ry 0 rz -180 deg; joints [-138.873, -59.458, -92.335, 44.737, 69.144, -19.431]
  Call Extruder(65.19540)
  MoveL 1776 to (-29.69, 36.18, 41.04) mm, rotated rx 180 ry 0 rz -180 deg; joints [-138.905, -59.464, -92.315, 44.709, 69.122, -19.431]
  MoveL 1777 to (-29.69, 36.18, 41.04) mm, rotated rx 180 ry 0 rz -180 deg; joints [-138.905, -59.464, -92.315, 44.709, 69.122, -19.431]
  Call Extruder(65.31047)
  MoveL 1778 to (-29.48, 36.14, 41.04) mm, rotated rx 180 ry 0 rz -180 deg; joints [-138.932, -59.469, -92.294, 44.685, 69.102, -19.433]
  MoveL 1779 to (-29.48, 36.14, 41.04) mm, rotated rx 180 ry 0 rz -180 deg; joints [-138.932, -59.469, -92.294, 44.685, 69.102, -19.433]
  Call Extruder(65.42509)
  MoveL 1780 to (-29.28, 36.09, 41.03) mm, rotated rx 180 ry 0 rz 180 deg; joints [-138.96, -59.475, -92.273, 44.662, 69.082, -19.434]
  MoveL 1781 to (-29.28, 36.09, 41.03) mm, rotated rx 180 ry 0 rz 180 deg; joints [-138.96, -59.475, -92.273, 44.662, 69.082, -19.434]
  Call Extruder(65.53926)
  MoveL 1782 to (-29.08, 36.05, 41.03) mm, rotated rx 180 ry 0 rz -180 deg; joints [-138.987, -59.48, -92.252, 44.638, 69.062, -19.436]
  MoveL 1783 to (-29.08, 36.05, 41.03) mm, rotated rx 180 ry 0 rz -180 deg; joints [-138.987, -59.48, -92.252, 44.638, 69.062, -19.436]
  Call Extruder(65.65298)
  MoveL 1784 to (-28.87, 36, 41.03) mm, rotated rx 180 ry 0 rz -180 deg; joints [-139.014, -59.486, -92.231, 44.615, 69.042, -19.438]
  MoveL 1785 to (-28.87, 36, 41.03) mm, rotated rx 180 ry 0 rz -180 deg; joints [-139.014, -59.486, -92.231, 44.615, 69.042, -19.438]
  Call Extruder(65.77840)
  MoveL 1786 to (-28.65, 35.96, 41.03) mm, rotated rx 180 ry 0 rz 180 deg; joints [-139.044, -59.492, -92.208, 44.589, 69.02, -19.44]
  MoveL 1787 to (-28.65, 35.96, 41.03) mm, rotated rx 180 ry 0 rz 180 deg; joints [-139.044, -59.492, -92.208, 44.589, 69.02, -19.44]
  Call Extruder(65.91538)
  MoveL 1788 to (-28.4, 35.91, 41.04) mm, rotated rx 180 ry 0 rz -180 deg; joints [-139.077, -59.499, -92.182, 44.561, 68.996, -19.443]
  MoveL 1789 to (-28.4, 35.91, 41.04) mm, rotated rx 180 ry 0 rz -180 deg; joints [-139.077, -59.499, -92.182, 44.561, 68.996, -19.443]
  Call Extruder(66.05174)
  MoveL 1790 to (-28.15, 35.86, 41.04) mm, rotated rx -180 ry 0 rz 180 deg; joints [-139.109, -59.506, -92.156, 44.534, 68.971, -19.445]
  MoveL 1791 to (-28.15, 35.86, 41.04) mm, rotated rx -180 ry 0 rz 180 deg; joints [-139.109, -59.506, -92.156, 44.534, 68.971, -19.445]
  Call Extruder(66.18750)
  MoveL 1792 to (-27.9, 35.81, 41.04) mm, rotated rx 180 ry 0 rz -180 deg; joints [-139.142, -59.513, -92.13, 44.506, 68.946, -19.448]
  MoveL 1793 to (-27.9, 35.81, 41.04) mm, rotated rx 180 ry 0 rz -180 deg; joints [-139.142, -59.513, -92.13, 44.506, 68.946, -19.448]
  Call Extruder(66.32265)
  MoveL 1794 to (-27.65, 35.76, 41.04) mm, rotated rx 180 ry 0 rz -180 deg; joints [-139.174, -59.52, -92.104, 44.478, 68.922, -19.45]
  MoveL 1795 to (-27.65, 35.76, 41.04) mm, rotated rx 180 ry 0 rz -180 deg; joints [-139.174, -59.52, -92.104, 44.478, 68.922, -19.45]
  Call Extruder(66.45718)
  MoveL 1796 to (-27.4, 35.71, 41.03) mm, rotated rx -180 ry 0 rz 180 deg; joints [-139.207, -59.526, -92.077, 44.45, 68.897, -19.453]
  MoveL 1797 to (-27.4, 35.71, 41.03) mm, rotated rx -180 ry 0 rz 180 deg; joints [-139.207, -59.526, -92.077, 44.45, 68.897, -19.453]
  Call Extruder(66.59111)
  MoveL 1798 to (-27.15, 35.66, 41.04) mm, rotated rx 180 ry 0 rz 180 deg; joints [-139.239, -59.533, -92.051, 44.423, 68.873, -19.456]
  MoveL 1799 to (-27.15, 35.66, 41.04) mm, rotated rx 180 ry 0 rz 180 deg; joints [-139.239, -59.533, -92.051, 44.423, 68.873, -19.456]
  Call Extruder(66.73897)
  MoveL 1800 to (-26.87, 35.61, 41.04) mm, rotated rx 180 ry 0 rz -180 deg; joints [-139.275, -59.541, -92.021, 44.393, 68.846, -19.459]
  MoveL 1801 to (-26.87, 35.61, 41.04) mm, rotated rx 180 ry 0 rz -180 deg; joints [-139.275, -59.541, -92.021, 44.393, 68.846, -19.459]
  Call Extruder(66.90071)
  MoveL 1802 to (-26.57, 35.56, 41.03) mm, rotated rx -180 ry 0 rz -180 deg; joints [-139.313, -59.55, -91.988, 44.361, 68.815, -19.464]
  MoveL 1803 to (-26.57, 35.56, 41.03) mm, rotated rx -180 ry 0 rz -180 deg; joints [-139.313, -59.55, -91.988, 44.361, 68.815, -19.464]
  Call Extruder(67.06171)
  MoveL 1804 to (-26.26, 35.51, 41.04) mm, rotated rx 180 ry 0 rz -180 deg; joints [-139.351, -59.559, -91.954, 44.329, 68.785, -19.468]
  MoveL 1805 to (-26.26, 35.51, 41.04) mm, rotated rx 180 ry 0 rz -180 deg; joints [-139.351, -59.559, -91.954, 44.329, 68.785, -19.468]
  Call Extruder(67.22199)
  MoveL 1806 to (-25.96, 35.46, 41.03) mm, rotated rx 180 ry 0 rz -180 deg; joints [-139.39, -59.568, -91.921, 44.297, 68.754, -19.473]
  MoveL 1807 to (-25.96, 35.46, 41.03) mm, rotated rx 180 ry 0 rz -180 deg; joints [-139.39, -59.568, -91.921, 44.297, 68.754, -19.473]
  Call Extruder(67.38154)
  MoveL 1808 to (-25.65, 35.42, 41.03) mm, rotated rx -180 ry 0 rz -180 deg; joints [-139.428, -59.577, -91.887, 44.265, 68.724, -19.477]
  MoveL 1809 to (-25.65, 35.42, 41.03) mm, rotated rx -180 ry 0 rz -180 deg; joints [-139.428, -59.577, -91.887, 44.265, 68.724, -19.477]
  Call Extruder(67.54036)
  MoveL 1810 to (-25.34, 35.37, 41.04) mm, rotated rx -180 ry 0 rz 180 deg; joints [-139.466, -59.586, -91.854, 44.233, 68.694, -19.482]
  MoveL 1811 to (-25.34, 35.37, 41.04) mm, rotated rx -180 ry 0 rz 180 deg; joints [-139.466, -59.586, -91.854, 44.233, 68.694, -19.482]
  Call Extruder(67.71903)
  MoveL 1812 to (-25, 35.32, 41.04) mm, rotated rx 180 ry 0 rz -180 deg; joints [-139.508, -59.596, -91.815, 44.198, 68.659, -19.487]
  MoveL 1813 to (-25, 35.32, 41.04) mm, rotated rx 180 ry 0 rz -180 deg; joints [-139.508, -59.596, -91.815, 44.198, 68.659, -19.487]
  Call Extruder(67.91748)
  MoveL 1814 to (-24.61, 35.27, 41.04) mm, rotated rx 180 ry 0 rz 180 deg; joints [-139.554, -59.608, -91.77, 44.16, 68.62, -19.495]
  MoveL 1815 to (-24.61, 35.27, 41.04) mm, rotated rx 180 ry 0 rz 180 deg; joints [-139.554, -59.608, -91.77, 44.16, 68.62, -19.495]
  Call Extruder(68.11505)
  MoveL 1816 to (-24.22, 35.23, 41.04) mm, rotated rx 180 ry 0 rz 180 deg; joints [-139.6, -59.62, -91.726, 44.123, 68.581, -19.502]
  MoveL 1817 to (-24.22, 35.23, 41.04) mm, rotated rx 180 ry 0 rz 180 deg; joints [-139.6, -59.62, -91.726, 44.123, 68.581, -19.502]
  Call Extruder(68.31176)
  MoveL 1818 to (-23.83, 35.18, 41.04) mm, rotated rx 180 ry 0 rz 180 deg; joints [-139.647, -59.632, -91.681, 44.085, 68.543, -19.509]
  MoveL 1819 to (-23.83, 35.18, 41.04) mm, rotated rx 180 ry 0 rz 180 deg; joints [-139.647, -59.632, -91.681, 44.085, 68.543, -19.509]
  Call Extruder(68.50760)
  MoveL 1820 to (-23.45, 35.14, 41.04) mm, rotated rx -180 ry 0 rz 180 deg; joints [-139.693, -59.644, -91.636, 44.047, 68.504, -19.517]
  MoveL 1821 to (-23.45, 35.14, 41.04) mm, rotated rx -180 ry 0 rz 180 deg; joints [-139.693, -59.644, -91.636, 44.047, 68.504, -19.517]
  Call Extruder(68.80299)
  MoveL 1822 to (-22.86, 35.09, 41.04) mm, rotated rx 180 ry 0 rz 180 deg; joints [-139.76, -59.663, -91.566, 43.993, 68.444, -19.53]
  MoveL 1823 to (-22.86, 35.09, 41.04) mm, rotated rx 180 ry 0 rz 180 deg; joints [-139.76, -59.663, -91.566, 43.993, 68.444, -19.53]
  Call Extruder(69.09705)
  MoveL 1824 to (-22.27, 35.05, 41.04) mm, rotated rx 180 ry 0 rz -180 deg; joints [-139.826, -59.682, -91.495, 43.94, 68.385, -19.544]
  MoveL 1825 to (-22.27, 35.05, 41.04) mm, rotated rx 180 ry 0 rz -180 deg; joints [-139.826, -59.682, -91.495, 43.94, 68.385, -19.544]
  Call Extruder(69.38978)
  MoveL 1826 to (-21.68, 35, 41.04) mm, rotated rx -180 ry 0 rz -180 deg; joints [-139.893, -59.701, -91.424, 43.886, 68.325, -19.558]
  MoveL 1827 to (-21.68, 35, 41.04) mm, rotated rx -180 ry 0 rz -180 deg; joints [-139.893, -59.701, -91.424, 43.886, 68.325, -19.558]
  Call Extruder(69.96323)
  MoveL 1828 to (-20.52, 34.95, 41.03) mm, rotated rx -180 ry 0 rz -180 deg; joints [-140.019, -59.741, -91.279, 43.788, 68.207, -19.589]
  MoveL 1829 to (-20.52, 34.95, 41.03) mm, rotated rx -180 ry 0 rz -180 deg; joints [-140.019, -59.741, -91.279, 43.788, 68.207, -19.589]
  Call Extruder(70.67720)
  MoveL 1830 to (-19.06, 34.91, 41.03) mm, rotated rx 180 ry 0 rz -180 deg; joints [-140.173, -59.791, -91.095, 43.669, 68.058, -19.631]
  Call Extruder(187.52394)
  MoveL 1831 to (219.06, 34.91, 41.04) mm, rotated rx 180 ry 0 rz 180 deg; joints [-155.896, -75.932, -48.39, 38.431, 41.073, -30.887]
  Call Extruder(187.95250)
  MoveL 1832 to (219.94, 34.93, 41.04) mm, rotated rx 180 ry 0 rz 180 deg; joints [-155.931, -76.031, -48.167, 38.474, 40.959, -30.97]
  MoveL 1833 to (219.94, 34.93, 41.04) mm, rotated rx 180 ry 0 rz 180 deg; joints [-155.931, -76.031, -48.167, 38.474, 40.959, -30.97]
  Call Extruder(188.52594)
  MoveL 1834 to (221.1, 34.97, 41.03) mm, rotated rx 180 ry 0 rz 180 deg; joints [-155.975, -76.165, -47.868, 38.536, 40.806, -31.085]
  MoveL 1835 to (221.1, 34.97, 41.03) mm, rotated rx 180 ry 0 rz 180 deg; joints [-155.975, -76.165, -47.868, 38.536, 40.806, -31.085]
  Call Extruder(188.96026)
  MoveL 1836 to (221.97, 35.02, 41.04) mm, rotated rx -180 ry 0 rz 180 deg; joints [-156.007, -76.267, -47.639, 38.586, 40.691, -31.174]
  MoveL 1837 to (221.97, 35.02, 41.04) mm, rotated rx -180 ry 0 rz 180 deg; joints [-156.007, -76.267, -47.639, 38.586, 40.691, -31.174]
  Call Extruder(189.25431)
  MoveL 1838 to (222.56, 35.07, 41.03) mm, rotated rx 180 ry 0 rz 180 deg; joints [-156.027, -76.336, -47.483, 38.623, 40.613, -31.236]
  MoveL 1839 to (222.56, 35.07, 41.03) mm, rotated rx 180 ry 0 rz 180 deg; joints [-156.027, -76.336, -47.483, 38.623, 40.613, -31.236]
  Call Extruder(189.54970)
  MoveL 1840 to (223.15, 35.11, 41.03) mm, rotated rx -180 ry 0 rz 180 deg; joints [-156.047, -76.406, -47.327, 38.659, 40.535, -31.299]
  MoveL 1841 to (223.15, 35.11, 41.03) mm, rotated rx -180 ry 0 rz 180 deg; joints [-156.047, -76.406, -47.327, 38.659, 40.535, -31.299]
  Call Extruder(189.79594)
  MoveL 1842 to (223.64, 35.16, 41.04) mm, rotated rx -180 ry 0 rz 180 deg; joints [-156.062, -76.465, -47.196, 38.691, 40.47, -31.353]
  MoveL 1843 to (223.64, 35.16, 41.04) mm, rotated rx -180 ry 0 rz 180 deg; joints [-156.062, -76.465, -47.196, 38.691, 40.47, -31.353]
  Call Extruder(189.99264)
  MoveL 1844 to (224.03, 35.21, 41.04) mm, rotated rx -180 ry 0 rz 180 deg; joints [-156.074, -76.512, -47.091, 38.719, 40.419, -31.397]
  MoveL 1845 to (224.03, 35.21, 41.04) mm, rotated rx -180 ry 0 rz 180 deg; joints [-156.074, -76.512, -47.091, 38.719, 40.419, -31.397]
  Call Extruder(190.19022)
  MoveL 1846 to (224.42, 35.25, 41.04) mm, rotated rx 180 ry 0 rz 180 deg; joints [-156.086, -76.559, -46.986, 38.746, 40.368, -31.442]
  MoveL 1847 to (224.42, 35.25, 41.04) mm, rotated rx 180 ry 0 rz 180 deg; joints [-156.086, -76.559, -46.986, 38.746, 40.368, -31.442]
  Call Extruder(190.38866)
  MoveL 1848 to (224.8, 35.3, 41.03) mm, rotated rx -180 ry 0 rz -180 deg; joints [-156.097, -76.606, -46.881, 38.774, 40.316, -31.487]
  MoveL 1849 to (224.8, 35.3, 41.03) mm, rotated rx -180 ry 0 rz -180 deg; joints [-156.097, -76.606, -46.881, 38.774, 40.316, -31.487]
  Call Extruder(190.58797)
  MoveL 1850 to (225.19, 35.34, 41.03) mm, rotated rx 180 ry 0 rz 180 deg; joints [-156.109, -76.653, -46.775, 38.801, 40.265, -31.531]
  MoveL 1851 to (225.19, 35.34, 41.03) mm, rotated rx 180 ry 0 rz 180 deg; joints [-156.109, -76.653, -46.775, 38.801, 40.265, -31.531]
  Call Extruder(190.74679)
  MoveL 1852 to (225.5, 35.39, 41.04) mm, rotated rx 180 ry 0 rz 180 deg; joints [-156.117, -76.691, -46.691, 38.825, 40.224, -31.569]
  MoveL 1853 to (225.5, 35.39, 41.04) mm, rotated rx 180 ry 0 rz 180 deg; joints [-156.117, -76.691, -46.691, 38.825, 40.224, -31.569]
  Call Extruder(190.90634)
  MoveL 1854 to (225.8, 35.44, 41.04) mm, rotated rx 180 ry 0 rz 180 deg; joints [-156.125, -76.729, -46.606, 38.85, 40.183, -31.606]
  MoveL 1855 to (225.8, 35.44, 41.04) mm, rotated rx 180 ry 0 rz 180 deg; joints [-156.125, -76.729, -46.606, 38.85, 40.183, -31.606]
  Call Extruder(191.06662)
  MoveL 1856 to (226.11, 35.49, 41.03) mm, rotated rx 180 ry 0 rz -180 deg; joints [-156.133, -76.767, -46.521, 38.874, 40.143, -31.643]
  MoveL 1857 to (226.11, 35.49, 41.03) mm, rotated rx 180 ry 0 rz -180 deg; joints [-156.133, -76.767, -46.521, 38.874, 40.143, -31.643]
  Call Extruder(191.22762)
  MoveL 1858 to (226.41, 35.54, 41.04) mm, rotated rx 180 ry 0 rz -180 deg; joints [-156.141, -76.805, -46.436, 38.898, 40.102, -31.681]
  MoveL 1859 to (226.41, 35.54, 41.04) mm, rotated rx 180 ry 0 rz -180 deg; joints [-156.141, -76.805, -46.436, 38.898, 40.102, -31.681]
  Call Extruder(191.38936)
  MoveL 1860 to (226.72, 35.59, 41.04) mm, rotated rx 180 ry 0 rz 180 deg; joints [-156.149, -76.844, -46.35, 38.923, 40.061, -31.719]
  MoveL 1861 to (226.72, 35.59, 41.04) mm, rotated rx 180 ry 0 rz 180 deg; joints [-156.149, -76.844, -46.35, 38.923, 40.061, -31.719]
  Call Extruder(191.55182)
  MoveL 1862 to (227.03, 35.63, 41.03) mm, rotated rx -180 ry 0 rz 180 deg; joints [-156.157, -76.882, -46.265, 38.948, 40.021, -31.757]
  MoveL 1863 to (227.03, 35.63, 41.03) mm, rotated rx -180 ry 0 rz 180 deg; joints [-156.157, -76.882, -46.265, 38.948, 40.021, -31.757]
  Call Extruder(191.68574)
  MoveL 1864 to (227.28, 35.68, 41.04) mm, rotated rx 180 ry 0 rz 180 deg; joints [-156.162, -76.914, -46.194, 38.969, 39.987, -31.789]
  MoveL 1865 to (227.28, 35.68, 41.04) mm, rotated rx 180 ry 0 rz 180 deg; joints [-156.162, -76.914, -46.194, 38.969, 39.987, -31.789]
  Call Extruder(191.82028)
  MoveL 1866 to (227.52, 35.73, 41.03) mm, rotated rx 180 ry 0 rz 180 deg; joints [-156.168, -76.946, -46.123, 38.991, 39.954, -31.822]
  MoveL 1867 to (227.52, 35.73, 41.03) mm, rotated rx 180 ry 0 rz 180 deg; joints [-156.168, -76.946, -46.123, 38.991, 39.954, -31.822]
  Call Extruder(191.95543)
  MoveL 1868 to (227.77, 35.78, 41.04) mm, rotated rx 180 ry 0 rz 180 deg; joints [-156.173, -76.978, -46.052, 39.013, 39.921, -31.855]
  MoveL 1869 to (227.77, 35.78, 41.04) mm, rotated rx 180 ry 0 rz 180 deg; joints [-156.173, -76.978, -46.052, 39.013, 39.921, -31.855]
  Call Extruder(192.09119)
  MoveL 1870 to (228.02, 35.83, 41.04) mm, rotated rx 180 ry 0 rz 180 deg; joints [-156.179, -77.01, -45.981, 39.035, 39.887, -31.887]
  MoveL 1871 to (228.02, 35.83, 41.04) mm, rotated rx 180 ry 0 rz 180 deg; joints [-156.179, -77.01, -45.981, 39.035, 39.887, -31.887]
  Call Extruder(192.22756)
  MoveL 1872 to (228.27, 35.88, 41.04) mm, rotated rx 180 ry 0 rz 180 deg; joints [-156.185, -77.042, -45.91, 39.058, 39.854, -31.92]
  MoveL 1873 to (228.27, 35.88, 41.04) mm, rotated rx 180 ry 0 rz 180 deg; joints [-156.185, -77.042, -45.91, 39.058, 39.854, -31.92]
  Call Extruder(192.36453)
  MoveL 1874 to (228.52, 35.93, 41.04) mm, rotated rx 180 ry 0 rz -180 deg; joints [-156.19, -77.074, -45.839, 39.08, 39.821, -31.953]
  MoveL 1875 to (228.52, 35.93, 41.04) mm, rotated rx 180 ry 0 rz -180 deg; joints [-156.19, -77.074, -45.839, 39.08, 39.821, -31.953]
  Call Extruder(192.50212)
  MoveL 1876 to (228.77, 35.98, 41.03) mm, rotated rx 180 ry 0 rz 180 deg; joints [-156.196, -77.106, -45.768, 39.102, 39.787, -31.986]
  MoveL 1877 to (228.77, 35.98, 41.03) mm, rotated rx 180 ry 0 rz 180 deg; joints [-156.196, -77.106, -45.768, 39.102, 39.787, -31.986]
  Call Extruder(192.61584)
  MoveL 1878 to (228.97, 36.03, 41.04) mm, rotated rx 180 ry 0 rz -180 deg; joints [-156.2, -77.132, -45.709, 39.121, 39.76, -32.014]
  MoveL 1879 to (228.97, 36.03, 41.04) mm, rotated rx 180 ry 0 rz -180 deg; joints [-156.2, -77.132, -45.709, 39.121, 39.76, -32.014]
  Call Extruder(192.73001)
  MoveL 1880 to (229.18, 36.07, 41.04) mm, rotated rx 180 ry 0 rz 180 deg; joints [-156.204, -77.159, -45.649, 39.14, 39.733, -32.042]
  MoveL 1881 to (229.18, 36.07, 41.04) mm, rotated rx 180 ry 0 rz 180 deg; joints [-156.204, -77.159, -45.649, 39.14, 39.733, -32.042]
  Call Extruder(192.84463)
  MoveL 1882 to (229.38, 36.12, 41.04) mm, rotated rx -180 ry 0 rz 180 deg; joints [-156.208, -77.186, -45.59, 39.16, 39.705, -32.07]
  MoveL 1883 to (229.38, 36.12, 41.04) mm, rotated rx -180 ry 0 rz 180 deg; joints [-156.208, -77.186, -45.59, 39.16, 39.705, -32.07]
  Call Extruder(192.95971)
  MoveL 1884 to (229.59, 36.16, 41.04) mm, rotated rx 180 ry 0 rz -180 deg; joints [-156.212, -77.212, -45.531, 39.179, 39.678, -32.097]
  MoveL 1885 to (229.59, 36.16, 41.04) mm, rotated rx 180 ry 0 rz -180 deg; joints [-156.212, -77.212, -45.531, 39.179, 39.678, -32.097]
  Call Extruder(193.08194)
  MoveL 1886 to (229.8, 36.22, 41.04) mm, rotated rx 180 ry 0 rz 180 deg; joints [-156.216, -77.241, -45.468, 39.201, 39.649, -32.128]
  MoveL 1887 to (229.8, 36.22, 41.04) mm, rotated rx 180 ry 0 rz 180 deg; joints [-156.216, -77.241, -45.468, 39.201, 39.649, -32.128]
  Call Extruder(193.21160)
  MoveL 1888 to (230.02, 36.28, 41.03) mm, rotated rx 180 ry 0 rz -180 deg; joints [-156.219, -77.271, -45.401, 39.225, 39.619, -32.162]
  MoveL 1889 to (230.02, 36.28, 41.03) mm, rotated rx 180 ry 0 rz -180 deg; joints [-156.219, -77.271, -45.401, 39.225, 39.619, -32.162]
  Call Extruder(193.34183)
  MoveL 1890 to (230.25, 36.35, 41.03) mm, rotated rx 180 ry 0 rz -180 deg; joints [-156.221, -77.301, -45.334, 39.249, 39.589, -32.195]
  MoveL 1891 to (230.25, 36.35, 41.03) mm, rotated rx 180 ry 0 rz -180 deg; joints [-156.221, -77.301, -45.334, 39.249, 39.589, -32.195]
  Call Extruder(193.47263)
  MoveL 1892 to (230.47, 36.42, 41.04) mm, rotated rx 180 ry 0 rz 180 deg; joints [-156.224, -77.331, -45.267, 39.274, 39.559, -32.229]
  MoveL 1893 to (230.47, 36.42, 41.04) mm, rotated rx 180 ry 0 rz 180 deg; joints [-156.224, -77.331, -45.267, 39.274, 39.559, -32.229]
  Call Extruder(193.60399)
  MoveL 1894 to (230.7, 36.49, 41.03) mm, rotated rx 180 ry 0 rz 180 deg; joints [-156.227, -77.362, -45.199, 39.299, 39.529, -32.263]
  MoveL 1895 to (230.7, 36.49, 41.03) mm, rotated rx 180 ry 0 rz 180 deg; joints [-156.227, -77.362, -45.199, 39.299, 39.529, -32.263]
  Call Extruder(193.72432)
  MoveL 1896 to (230.9, 36.55, 41.04) mm, rotated rx 180 ry 0 rz 180 deg; joints [-156.229, -77.39, -45.138, 39.322, 39.502, -32.295]
  MoveL 1897 to (230.9, 36.55, 41.04) mm, rotated rx 180 ry 0 rz 180 deg; joints [-156.229, -77.39, -45.138, 39.322, 39.502, -32.295]
  Call Extruder(193.84516)
  MoveL 1898 to (231.1, 36.62, 41.03) mm, rotated rx 180 ry 0 rz -180 deg; joints [-156.231, -77.418, -45.076, 39.345, 39.474, -32.326]
  MoveL 1899 to (231.1, 36.62, 41.03) mm, rotated rx 180 ry 0 rz -180 deg; joints [-156.231, -77.418, -45.076, 39.345, 39.474, -32.326]
  Call Extruder(193.96651)
  MoveL 1900 to (231.3, 36.68, 41.04) mm, rotated rx -180 ry 0 rz 180 deg; joints [-156.234, -77.445, -45.014, 39.368, 39.447, -32.358]
  MoveL 1901 to (231.3, 36.68, 41.04) mm, rotated rx -180 ry 0 rz 180 deg; joints [-156.234, -77.445, -45.014, 39.368, 39.447, -32.358]
  Call Extruder(194.08838)
  MoveL 1902 to (231.51, 36.75, 41.04) mm, rotated rx 180 ry 0 rz 180 deg; joints [-156.236, -77.473, -44.953, 39.391, 39.42, -32.389]
  MoveL 1903 to (231.51, 36.75, 41.04) mm, rotated rx 180 ry 0 rz 180 deg; joints [-156.236, -77.473, -44.953, 39.391, 39.42, -32.389]
  Call Extruder(194.21076)
  MoveL 1904 to (231.71, 36.82, 41.03) mm, rotated rx -180 ry 0 rz 180 deg; joints [-156.238, -77.501, -44.891, 39.415, 39.392, -32.421]
  MoveL 1905 to (231.71, 36.82, 41.03) mm, rotated rx -180 ry 0 rz 180 deg; joints [-156.238, -77.501, -44.891, 39.415, 39.392, -32.421]
  Call Extruder(194.33365)
  MoveL 1906 to (231.91, 36.88, 41.03) mm, rotated rx -180 ry 0 rz 180 deg; joints [-156.24, -77.529, -44.829, 39.438, 39.365, -32.453]
  MoveL 1907 to (231.91, 36.88, 41.03) mm, rotated rx -180 ry 0 rz 180 deg; joints [-156.24, -77.529, -44.829, 39.438, 39.365, -32.453]
  Call Extruder(194.51082)
  MoveL 1908 to (232.19, 37, 41.04) mm, rotated rx 180 ry 0 rz 180 deg; joints [-156.241, -77.57, -44.739, 39.475, 39.327, -32.501]
  MoveL 1909 to (232.19, 37, 41.04) mm, rotated rx 180 ry 0 rz 180 deg; joints [-156.241, -77.57, -44.739, 39.475, 39.327, -32.501]
  Call Extruder(194.72368)
  MoveL 1910 to (232.53, 37.15, 41.04) mm, rotated rx -180 ry 0 rz 180 deg; joints [-156.24, -77.618, -44.632, 39.522, 39.282, -32.561]
  MoveL 1911 to (232.53, 37.15, 41.04) mm, rotated rx -180 ry 0 rz 180 deg; joints [-156.24, -77.618, -44.632, 39.522, 39.282, -32.561]
  Call Extruder(194.91775)
  MoveL 1912 to (232.83, 37.29, 41.03) mm, rotated rx 180 ry 0 rz 180 deg; joints [-156.24, -77.662, -44.534, 39.564, 39.241, -32.615]
  MoveL 1913 to (232.83, 37.29, 41.03) mm, rotated rx 180 ry 0 rz 180 deg; joints [-156.24, -77.662, -44.534, 39.564, 39.241, -32.615]
  Call Extruder(195.11861)
  MoveL 1914 to (233.13, 37.45, 41.04) mm, rotated rx 180 ry 0 rz 180 deg; joints [-156.238, -77.708, -44.434, 39.609, 39.199, -32.672]
  MoveL 1915 to (233.13, 37.45, 41.04) mm, rotated rx 180 ry 0 rz 180 deg; joints [-156.238, -77.708, -44.434, 39.609, 39.199, -32.672]
  Call Extruder(195.32676)
  MoveL 1916 to (233.44, 37.62, 41.04) mm, rotated rx 180 ry 0 rz 180 deg; joints [-156.234, -77.755, -44.33, 39.659, 39.158, -32.734]
  MoveL 1917 to (233.44, 37.62, 41.04) mm, rotated rx 180 ry 0 rz 180 deg; joints [-156.234, -77.755, -44.33, 39.659, 39.158, -32.734]
  Call Extruder(195.53571)
  MoveL 1918 to (233.75, 37.8, 41.04) mm, rotated rx 180 ry 0 rz 180 deg; joints [-156.23, -77.802, -44.227, 39.708, 39.116, -32.795]
  MoveL 1919 to (233.75, 37.8, 41.04) mm, rotated rx 180 ry 0 rz 180 deg; joints [-156.23, -77.802, -44.227, 39.708, 39.116, -32.795]
  Call Extruder(195.74544)
  MoveL 1920 to (234.05, 37.98, 41.04) mm, rotated rx 180 ry 0 rz -180 deg; joints [-156.226, -77.849, -44.123, 39.758, 39.075, -32.856]
  MoveL 1921 to (234.05, 37.98, 41.04) mm, rotated rx 180 ry 0 rz -180 deg; joints [-156.226, -77.849, -44.123, 39.758, 39.075, -32.856]
  Call Extruder(195.86398)
  MoveL 1922 to (234.22, 38.08, 41.03) mm, rotated rx 180 ry 0 rz -180 deg; joints [-156.224, -77.875, -44.064, 39.786, 39.051, -32.891]
  MoveL 1923 to (234.22, 38.08, 41.03) mm, rotated rx 180 ry 0 rz -180 deg; joints [-156.224, -77.875, -44.064, 39.786, 39.051, -32.891]
  Call Extruder(196.19680)
  MoveL 1924 to (234.68, 38.41, 41.03) mm, rotated rx 180 ry 0 rz -180 deg; joints [-156.212, -77.949, -43.902, 39.872, 38.99, -32.993]
  MoveL 1925 to (234.68, 38.41, 41.03) mm, rotated rx 180 ry 0 rz -180 deg; joints [-156.212, -77.949, -43.902, 39.872, 38.99, -32.993]
  Call Extruder(196.53081)
  MoveL 1926 to (235.13, 38.73, 41.04) mm, rotated rx 180 ry 0 rz -180 deg; joints [-156.201, -78.022, -43.741, 39.958, 38.928, -33.096]
  MoveL 1927 to (235.13, 38.73, 41.04) mm, rotated rx 180 ry 0 rz -180 deg; joints [-156.201, -78.022, -43.741, 39.958, 38.928, -33.096]
  Call Extruder(196.69838)
  MoveL 1928 to (235.35, 38.9, 41.04) mm, rotated rx -180 ry 0 rz 180 deg; joints [-156.195, -78.059, -43.659, 40.001, 38.897, -33.147]
  Call Extruder(197.52772)
  MoveL 1929 to (236.39, 39.81, 41.04) mm, rotated rx -180 ry 0 rz 180 deg; joints [-156.154, -78.238, -43.266, 40.227, 38.756, -33.41]
  Call Extruder(198.15878)
  MoveL 1930 to (237.09, 40.59, 41.03) mm, rotated rx -180 ry 0 rz 180 deg; joints [-156.111, -78.369, -42.978, 40.411, 38.66, -33.617]
  MoveL 1931 to (237.09, 40.59, 41.03) mm, rotated rx -180 ry 0 rz 180 deg; joints [-156.111, -78.369, -42.978, 40.411, 38.66, -33.617]
  Call Extruder(198.35639)
  MoveL 1932 to (237.3, 40.85, 41.04) mm, rotated rx 180 ry 0 rz 180 deg; joints [-156.097, -78.41, -42.888, 40.47, 38.631, -33.683]
  Call Extruder(198.69040)
  MoveL 1933 to (237.63, 41.3, 41.03) mm, rotated rx -180 ry 0 rz 180 deg; joints [-156.069, -78.476, -42.742, 40.571, 38.586, -33.794]
  MoveL 1934 to (237.63, 41.3, 41.03) mm, rotated rx -180 ry 0 rz 180 deg; joints [-156.069, -78.476, -42.742, 40.571, 38.586, -33.794]
  Call Extruder(199.02322)
  MoveL 1935 to (237.96, 41.75, 41.03) mm, rotated rx 180 ry 0 rz -180 deg; joints [-156.042, -78.543, -42.596, 40.673, 38.54, -33.906]
  MoveL 1936 to (237.96, 41.75, 41.03) mm, rotated rx 180 ry 0 rz -180 deg; joints [-156.042, -78.543, -42.596, 40.673, 38.54, -33.906]
  Call Extruder(199.20245)
  MoveL 1937 to (238.13, 41.99, 41.04) mm, rotated rx -180 ry 0 rz 180 deg; joints [-156.027, -78.579, -42.517, 40.728, 38.516, -33.966]
  MoveL 1938 to (238.13, 41.99, 41.04) mm, rotated rx -180 ry 0 rz 180 deg; joints [-156.027, -78.579, -42.517, 40.728, 38.516, -33.966]
  Call Extruder(199.41057)
  MoveL 1939 to (238.31, 42.3, 41.03) mm, rotated rx 180 ry 0 rz 180 deg; joints [-156.006, -78.619, -42.431, 40.793, 38.492, -34.037]
  MoveL 1940 to (238.31, 42.3, 41.03) mm, rotated rx 180 ry 0 rz 180 deg; joints [-156.006, -78.619, -42.431, 40.793, 38.492, -34.037]
  Call Extruder(199.61791)
  MoveL 1941 to (238.49, 42.6, 41.03) mm, rotated rx 180 ry 0 rz 180 deg; joints [-155.986, -78.658, -42.344, 40.859, 38.468, -34.107]
  MoveL 1942 to (238.49, 42.6, 41.03) mm, rotated rx 180 ry 0 rz 180 deg; joints [-155.986, -78.658, -42.344, 40.859, 38.468, -34.107]
  Call Extruder(199.82447)
  MoveL 1943 to (238.66, 42.91, 41.03) mm, rotated rx 180 ry 0 rz 180 deg; joints [-155.966, -78.698, -42.257, 40.925, 38.444, -34.178]
  MoveL 1944 to (238.66, 42.91, 41.03) mm, rotated rx 180 ry 0 rz 180 deg; joints [-155.966, -78.698, -42.257, 40.925, 38.444, -34.178]
  Call Extruder(200.03025)
  MoveL 1945 to (238.84, 43.21, 41.04) mm, rotated rx -180 ry 0 rz 180 deg; joints [-155.946, -78.737, -42.171, 40.99, 38.419, -34.249]
  MoveL 1946 to (238.84, 43.21, 41.04) mm, rotated rx -180 ry 0 rz 180 deg; joints [-155.946, -78.737, -42.171, 40.99, 38.419, -34.249]
  Call Extruder(200.18856)
  MoveL 1947 to (238.94, 43.46, 41.04) mm, rotated rx -180 ry 0 rz -180 deg; joints [-155.927, -78.765, -42.11, 41.042, 38.405, -34.302]
  MoveL 1948 to (238.94, 43.46, 41.04) mm, rotated rx -180 ry 0 rz -180 deg; joints [-155.927, -78.765, -42.11, 41.042, 38.405, -34.302]
  Call Extruder(200.34626)
  MoveL 1949 to (239.05, 43.71, 41.03) mm, rotated rx -180 ry 0 rz 180 deg; joints [-155.909, -78.793, -42.049, 41.093, 38.39, -34.356]
  MoveL 1950 to (239.05, 43.71, 41.03) mm, rotated rx -180 ry 0 rz 180 deg; joints [-155.909, -78.793, -42.049, 41.093, 38.39, -34.356]
  Call Extruder(200.51634)
  MoveL 1951 to (239.17, 43.98, 41.04) mm, rotated rx 180 ry 0 rz 180 deg; joints [-155.89, -78.823, -41.983, 41.149, 38.374, -34.414]
  MoveL 1952 to (239.17, 43.98, 41.04) mm, rotated rx 180 ry 0 rz 180 deg; joints [-155.89, -78.823, -41.983, 41.149, 38.374, -34.414]
  Call Extruder(200.69866)
  MoveL 1953 to (239.29, 44.27, 41.03) mm, rotated rx -180 ry 0 rz -180 deg; joints [-155.869, -78.855, -41.913, 41.209, 38.357, -34.477]
  MoveL 1954 to (239.29, 44.27, 41.03) mm, rotated rx -180 ry 0 rz -180 deg; joints [-155.869, -78.855, -41.913, 41.209, 38.357, -34.477]
  Call Extruder(200.88022)
  MoveL 1955 to (239.41, 44.56, 41.04) mm, rotated rx 180 ry 0 rz 180 deg; joints [-155.847, -78.888, -41.842, 41.269, 38.34, -34.54]
  MoveL 1956 to (239.41, 44.56, 41.04) mm, rotated rx 180 ry 0 rz 180 deg; joints [-155.847, -78.888, -41.842, 41.269, 38.34, -34.54]
  Call Extruder(200.93707)
  MoveL 1957 to (239.44, 44.66, 41.03) mm, rotated rx -180 ry 0 rz -180 deg; joints [-155.84, -78.897, -41.822, 41.288, 38.336, -34.559]
  MoveL 1958 to (239.44, 44.66, 41.03) mm, rotated rx -180 ry 0 rz -180 deg; joints [-155.84, -78.897, -41.822, 41.288, 38.336, -34.559]
  Call Extruder(201.05031)
  MoveL 1959 to (239.5, 44.85, 41.04) mm, rotated rx 180 ry 0 rz 180 deg; joints [-155.826, -78.916, -41.781, 41.326, 38.328, -34.598]
  MoveL 1960 to (239.5, 44.85, 41.04) mm, rotated rx 180 ry 0 rz 180 deg; joints [-155.826, -78.916, -41.781, 41.326, 38.328, -34.598]
  Call Extruder(201.16311)
  MoveL 1961 to (239.56, 45.03, 41.04) mm, rotated rx 180 ry 0 rz 180 deg; joints [-155.811, -78.934, -41.74, 41.363, 38.319, -34.636]
  MoveL 1962 to (239.56, 45.03, 41.04) mm, rotated rx 180 ry 0 rz 180 deg; joints [-155.811, -78.934, -41.74, 41.363, 38.319, -34.636]
  Call Extruder(201.27546)
  MoveL 1963 to (239.62, 45.22, 41.03) mm, rotated rx 180 ry 0 rz -180 deg; joints [-155.797, -78.953, -41.699, 41.401, 38.311, -34.675]
  MoveL 1964 to (239.62, 45.22, 41.03) mm, rotated rx 180 ry 0 rz -180 deg; joints [-155.797, -78.953, -41.699, 41.401, 38.311, -34.675]
  Call Extruder(201.38737)
  MoveL 1965 to (239.68, 45.41, 41.03) mm, rotated rx -180 ry 0 rz 180 deg; joints [-155.783, -78.972, -41.658, 41.438, 38.302, -34.714]
  MoveL 1966 to (239.68, 45.41, 41.03) mm, rotated rx -180 ry 0 rz 180 deg; joints [-155.783, -78.972, -41.658, 41.438, 38.302, -34.714]
  Call Extruder(201.50878)
  MoveL 1967 to (239.75, 45.62, 41.03) mm, rotated rx 180 ry 0 rz 180 deg; joints [-155.767, -78.992, -41.613, 41.479, 38.293, -34.756]
  MoveL 1968 to (239.75, 45.62, 41.03) mm, rotated rx 180 ry 0 rz 180 deg; joints [-155.767, -78.992, -41.613, 41.479, 38.293, -34.756]
  Call Extruder(201.63957)
  MoveL 1969 to (239.81, 45.84, 41.03) mm, rotated rx 180 ry 0 rz 180 deg; joints [-155.75, -79.014, -41.566, 41.524, 38.284, -34.801]
  MoveL 1970 to (239.81, 45.84, 41.03) mm, rotated rx 180 ry 0 rz 180 deg; joints [-155.75, -79.014, -41.566, 41.524, 38.284, -34.801]
  Call Extruder(201.76979)
  MoveL 1971 to (239.88, 46.06, 41.04) mm, rotated rx 180 ry 0 rz 180 deg; joints [-155.733, -79.036, -41.519, 41.568, 38.274, -34.847]
  MoveL 1972 to (239.88, 46.06, 41.04) mm, rotated rx 180 ry 0 rz 180 deg; joints [-155.733, -79.036, -41.519, 41.568, 38.274, -34.847]
  Call Extruder(201.89946)
  MoveL 1973 to (239.95, 46.29, 41.04) mm, rotated rx 180 ry 0 rz 180 deg; joints [-155.715, -79.057, -41.471, 41.613, 38.265, -34.892]
  MoveL 1974 to (239.95, 46.29, 41.04) mm, rotated rx 180 ry 0 rz 180 deg; joints [-155.715, -79.057, -41.471, 41.613, 38.265, -34.892]
  Call Extruder(202.02855)
  MoveL 1975 to (240.02, 46.51, 41.04) mm, rotated rx 180 ry 0 rz 180 deg; joints [-155.698, -79.079, -41.424, 41.657, 38.256, -34.938]
  MoveL 1976 to (240.02, 46.51, 41.04) mm, rotated rx 180 ry 0 rz 180 deg; joints [-155.698, -79.079, -41.424, 41.657, 38.256, -34.938]
  Call Extruder(202.14360)
  MoveL 1977 to (240.06, 46.72, 41.04) mm, rotated rx -180 ry 0 rz -180 deg; joints [-155.682, -79.097, -41.385, 41.696, 38.249, -34.977]
  MoveL 1978 to (240.06, 46.72, 41.04) mm, rotated rx -180 ry 0 rz -180 deg; joints [-155.682, -79.097, -41.385, 41.696, 38.249, -34.977]
  Call Extruder(202.25820)
  MoveL 1979 to (240.11, 46.92, 41.04) mm, rotated rx -180 ry 0 rz -180 deg; joints [-155.665, -79.115, -41.346, 41.736, 38.243, -35.017]
  MoveL 1980 to (240.11, 46.92, 41.04) mm, rotated rx -180 ry 0 rz -180 deg; joints [-155.665, -79.115, -41.346, 41.736, 38.243, -35.017]
  Call Extruder(202.37235)
  MoveL 1981 to (240.15, 47.12, 41.04) mm, rotated rx 180 ry 0 rz 180 deg; joints [-155.649, -79.132, -41.308, 41.775, 38.237, -35.056]
  MoveL 1982 to (240.15, 47.12, 41.04) mm, rotated rx 180 ry 0 rz 180 deg; joints [-155.649, -79.132, -41.308, 41.775, 38.237, -35.056]
  Call Extruder(202.48605)
  MoveL 1983 to (240.2, 47.33, 41.04) mm, rotated rx 180 ry 0 rz 180 deg; joints [-155.633, -79.15, -41.269, 41.815, 38.231, -35.096]
  MoveL 1984 to (240.2, 47.33, 41.04) mm, rotated rx 180 ry 0 rz 180 deg; joints [-155.633, -79.15, -41.269, 41.815, 38.231, -35.096]
  Call Extruder(202.61146)
  MoveL 1985 to (240.24, 47.55, 41.04) mm, rotated rx 180 ry 0 rz 180 deg; joints [-155.614, -79.17, -41.226, 41.858, 38.224, -35.139]
  MoveL 1986 to (240.24, 47.55, 41.04) mm, rotated rx 180 ry 0 rz 180 deg; joints [-155.614, -79.17, -41.226, 41.858, 38.224, -35.139]
  Call Extruder(202.74844)
  MoveL 1987 to (240.29, 47.8, 41.04) mm, rotated rx 180 ry 0 rz 180 deg; joints [-155.594, -79.191, -41.18, 41.906, 38.217, -35.187]
  MoveL 1988 to (240.29, 47.8, 41.04) mm, rotated rx 180 ry 0 rz 180 deg; joints [-155.594, -79.191, -41.18, 41.906, 38.217, -35.187]
  Call Extruder(202.88480)
  MoveL 1989 to (240.34, 48.05, 41.03) mm, rotated rx 180 ry 0 rz 180 deg; joints [-155.574, -79.212, -41.134, 41.953, 38.21, -35.235]
  MoveL 1990 to (240.34, 48.05, 41.03) mm, rotated rx 180 ry 0 rz 180 deg; joints [-155.574, -79.212, -41.134, 41.953, 38.21, -35.235]
  Call Extruder(203.02056)
  MoveL 1991 to (240.39, 48.3, 41.03) mm, rotated rx 180 ry 0 rz -180 deg; joints [-155.554, -79.233, -41.088, 42.001, 38.203, -35.283]
  MoveL 1992 to (240.39, 48.3, 41.03) mm, rotated rx 180 ry 0 rz -180 deg; joints [-155.554, -79.233, -41.088, 42.001, 38.203, -35.283]
  Call Extruder(203.15571)
